(*=======================================================*)
	INIT:
		IF fb_state_entry.E THEN
			fb_ton_wz.IN := FALSE;
			fb_ton_uez.IN := FALSE;
			fb_ton_quitt.IN := FALSE;
			st_ctrl_out.b_fehler := FALSE;
			st_ctrl_out.b_bereit := FALSE;
			st_ctrl_out.b_fertig := FALSE;
			st_ctrl_out.b_kontroller_start := FALSE;
			zyl_wt_zentrierer_tisch.st_ctrl.in.b_einfahren := FALSE;
			zyl_wt_zentrierer_tisch.st_ctrl.in.b_ausfahren := FALSE;
			zyl_wt_zentrierer_tisch.st_ctrl.in.b_luftlos := FALSE;
			axis_transport_wt_achse.st_ctrl.in.b_start := FALSE;
			axis_z_achse.st_ctrl.in.b_start := FALSE;
			stueckzahlen.st_ctrl.in.b_gutteil_produziert := FALSE;
			sm_wt_hat_beladepos_nicht_verlassen := FALSE;
			sm_tagnummer_ungueltig := FALSE;
			sm_wt_hat_kein_tag := FALSE;
			sm_tagreader_nicht_fertig := FALSE;
			sm_keine_bandfreigabe := FALSE;
			bm_abfrage_wt_auf_beladepos := FALSE;
			bm_warte_auf_wt_an_stopper := FALSE;
			balluff_tag_reader.st_ctrl.in.b_start_lesen := FALSE;
			balluff_tag_reader.st_ctrl.in.b_start_schreiben := FALSE;
			zyl_Indexier_Bestueckpos.st_ctrl.in.b_ausfahren := FALSE;
			zyl_Indexier_Bestueckpos.st_ctrl.in.b_einfahren := FALSE;
			bMerkerSchrittketteKommtVonInit := TRUE;
		END_IF

		(*-----------------------Weiterschaltbedingungen----------------------------*)
		IF st_ctrl_in.b_init THEN
			zyl_wt_zentrierer_tisch.st_ctrl.in.b_quittieren := FALSE;
			zyl_Indexier_Bestueckpos.st_ctrl.in.b_quittieren := FALSE;
			fb_state_entry.i16_next_step := 20;
		END_IF

(*=======================================================*)
	20: fb_state_entry.s_debugtext := 'Initialisierung: Stopper an Bestücktisch ausfahren und Zentrierer einfahren';

		(*-----------------------Weiterschaltbedingungen----------------------------*)
		IF e_wt_im_aktionsfeld THEN
			fb_state_entry.i16_next_step := 25;
		ELSE
			fb_state_entry.i16_next_step := 22;
		END_IF

(*=======================================================*)
	22: fb_state_entry.s_debugtext := 'Initialisierung: Stopper an Bestücktisch ausfahren und Zentrierer einfahren';

		IF fb_state_entry.E THEN
			zyl_wt_zentrierer_tisch.st_ctrl.in.b_einfahren := TRUE;
		END_IF

		(*-----------------------Weiterschaltbedingungen----------------------------*)
		IF  zyl_wt_zentrierer_tisch.st_ctrl.out.b_eingefahren THEN
			zyl_wt_zentrierer_tisch.st_ctrl.in.b_einfahren := FALSE;
			fb_state_entry.i16_next_step := 30;
		END_IF

(*=======================================================*)
	25: fb_state_entry.s_debugtext := 'Initialisierung: Stopper an Bestücktisch ausfahren und Zentrierer einfahren';

		IF fb_state_entry.E THEN
			zyl_wt_zentrierer_tisch.st_ctrl.in.b_ausfahren := TRUE;
		END_IF

		(*-----------------------Weiterschaltbedingungen----------------------------*)
		IF  zyl_wt_zentrierer_tisch.st_ctrl.out.b_ausgefahren THEN
			zyl_wt_zentrierer_tisch.st_ctrl.in.b_ausfahren := FALSE;
			fb_state_entry.i16_next_step := 30;
		END_IF

(*=======================================================*)
	30: fb_state_entry.s_debugtext := 'Indexierzylinder wieder einfahren';

		IF fb_state_entry.E THEN
			zyl_Indexier_Bestueckpos.st_ctrl.in.b_ausfahren:= TRUE;
		END_IF

		(*-----------------------Weiterschaltbedingungen----------------------------*)
		IF zyl_Indexier_Bestueckpos.st_ctrl.out.b_ausgefahren THEN
			zyl_Indexier_Bestueckpos.st_ctrl.in.b_ausfahren:= FALSE;
			fb_state_entry.i16_next_step := 35;
		END_IF

(*=======================================================*)
	35: fb_state_entry.s_debugtext := 'warten auf Achse bereit';

		(*-----------------------Weiterschaltbedingungen----------------------------*)
		IF	axis_transport_wt_achse.st_ctrl.out.b_bereit AND
			NOT axis_transport_wt_achse.st_ctrl.in.b_start THEN
			fb_state_entry.i16_next_step := 40;
		END_IF

(*=======================================================*)
	40: fb_state_entry.s_debugtext := 'Fahre Achse wieder zurück';

		IF fb_state_entry.E THEN
			ST_WT_Transport_Achse.lr_Achspos_in:=gst_datensatz.st_md.st_md_transport_wt_achse.lr_startposition;
			ST_WT_Transport_Achse.lr_Velo_in:= gst_datensatz.st_md.r_geschwindigkeit_achse_transport;
			ST_WT_Transport_Achse.enu_cmd_in:=MOVE_ABSOLUTE;
			axis_transport_wt_achse.st_ctrl.in.b_start := TRUE;
		END_IF

		(*-----------------------Weiterschaltbedingungen----------------------------*)
		IF  axis_transport_wt_achse.st_ctrl.out.b_busy THEN
			axis_transport_wt_achse.st_ctrl.in.b_start := FALSE;
			fb_state_entry.i16_next_step := 50;
		END_IF

(*=======================================================*)
	50: fb_state_entry.s_debugtext := 'warten auf Achse hinten fertig';

		(*-----------------------Weiterschaltbedingungen----------------------------*)
		IF	axis_transport_wt_achse.st_ctrl.out.b_fertig  THEN
			fb_state_entry.i16_next_step := BEREIT;
		END_IF

(*=======================================================*)
	BEREIT:	fb_state_entry.s_debugtext := 'Warte auf Start von Kontroller';

		IF fb_state_entry.E THEN
			st_ctrl_out.b_bereit := TRUE;
			st_ctrl_out.b_fertig := TRUE;
			stueckzahlen.st_ctrl.in.b_gutteil_produziert := FALSE;
		END_IF

		(*-----------------------Weiterschaltbedingungen----------------------------*)
		IF st_config.b_station_aktiv OR st_config.b_station_in_simulation THEN

		(* WT Transport aktiv oder in Simulation *)
			IF 	st_ctrl_in.b_start  AND
				((NOT ST_Virtuelle_Masterachse.b_merker_bandende_links  AND
 				NOT ST_Virtuelle_Masterachse.b_merker_bandende_rechts) OR
				gst_datensatz.st_md.b_auto_Bandwechsel) THEN
			(* WT Transport gestartet *)
				st_ctrl_out.b_fertig := FALSE;
				fb_ton_wz.IN := FALSE;
				st_ctrl_out.b_kontroller_start := TRUE;
				(* Abfrage, ob Schrittkette von Init kommt und ob WT auf Beladepos ist *)
				IF bMerkerSchrittketteKommtVonInit AND
					e_wt_auf_beladepos THEN
					fb_state_entry.i16_next_step := 150;	(* WT auslesen und prüfen, ob dieser schon bestückt wurde *)
				ELSE
					fb_state_entry.i16_next_step := 110;
				END_IF
			END_IF

		(* WT-Transport nicht aktiv  *)
		ELSE
			IF fb_r_trig_start.Q THEN
				(* Nur Z-Achse gestartet *)
				st_ctrl_out.b_fertig := FALSE;
				fb_ton_wz.IN := FALSE;
				fb_state_entry.i16_next_step := 500;
			END_IF
		END_IF

		IF fb_state_entry.X THEN
			bMerkerSchrittketteKommtVonInit := FALSE;
		END_IF

(*=======================================================*)
	110: fb_state_entry.s_debugtext := 'WT-Abfrage auf Beladeposition';

		IF fb_state_entry.E THEN
			bm_abfrage_wt_auf_beladepos := TRUE;
		END_IF

		(*-----------------------Weiterschaltbedingungen----------------------------*)
		IF e_wt_im_aktionsfeld THEN
			(* Ein WT ist anwesend zum rausschicken *)
			IF NOT ST_WT_Transport_Abgabe.e_wt_auf_abgabepos THEN
				(* Erst wenn kein Stau vorhanden ist, dann wird der WT weiter gelassen *)
				fb_state_entry.i16_next_step := 115;
			END_IF
		ELSE	(* Kein WT da, deshalb einen holen *)
			fb_state_entry.i16_next_step := 130;
		END_IF

		IF fb_state_entry.X THEN
			bm_abfrage_wt_auf_beladepos := FALSE;
			st_ctrl_out.b_kontroller_start := FALSE;
		END_IF

(*=======================================================*)
	115: fb_state_entry.s_debugtext := 'Indexierzylinder Bestückposition ausfahren (WT festhalten)';

		IF fb_state_entry.E THEN
			zyl_Indexier_Bestueckpos.st_ctrl.in.b_einfahren:= TRUE;
		END_IF

		(*-----------------------Weiterschaltbedingungen----------------------------*)
		IF zyl_Indexier_Bestueckpos.st_ctrl.out.b_eingefahren THEN
			zyl_Indexier_Bestueckpos.st_ctrl.in.b_einfahren:= FALSE;
			fb_state_entry.i16_next_step := 120;
		END_IF

(*=======================================================*)
	120: fb_state_entry.s_debugtext := 'WT-Zentrierer einfahren';

		IF fb_state_entry.E THEN
			zyl_wt_zentrierer_tisch.st_ctrl.in.b_einfahren := TRUE;
			fb_Zentrierer_einfahren(b_start:= TRUE, t_zeit=> );
		END_IF

		(*-----------------------Weiterschaltbedingungen----------------------------*)
		IF zyl_wt_zentrierer_tisch.st_ctrl.out.b_eingefahren THEN
			zyl_wt_zentrierer_tisch.st_ctrl.in.b_einfahren := FALSE;
			fb_Zentrierer_einfahren(b_start:= FALSE, t_zeit=>t_Zentrierer_einfahren);
			fb_state_entry.i16_next_step := 130;
		END_IF

(*=======================================================*)
	130: fb_state_entry.s_debugtext := 'WT ist auf Warteposition und mit Indexierzylinder fixiert, wenn 2 Sekunden kein WT aus der vorherigen Zelle kommt wird der WT weitergeschickt';

		IF fb_state_entry.E THEN
			bm_abfrage_wt_auf_wartepos := TRUE;
		END_IF

		(*-----------------------Weiterschaltbedingungen----------------------------*)
		IF ST_WT_Transport_Warteposition_1700.e_wt_auf_wartepos_1700 AND
			 zyl_Indexier_Einlauf.st_ctrl.out.b_eingefahren AND
			ST_WT_Transport_Warteposition_1700.b_helpStartAchse AND
			zyl_wt_stopper_tisch.st_ctrl.out.b_eingefahren THEN
			fb_state_entry.i16_next_step := 135;
		ELSIF fb_state_entry.fb_ton_Step.ET >= T#2S AND
			 zyl_Indexier_Bestueckpos.st_ctrl.out.b_eingefahren THEN
			fb_state_entry.i16_next_step := 132;
		END_IF

(*=======================================================*)
	132: fb_state_entry.s_debugtext := 'Warten bis kein WT mehr auf der Abgabeposition steht';

		(*-----------------------Weiterschaltbedingungen----------------------------*)
		IF NOT ST_WT_Transport_Abgabe.e_wt_auf_abgabepos THEN
			fb_state_entry.i16_next_step := 135;
		END_IF

(*=======================================================*)
	135: fb_state_entry.s_debugtext := 'warten auf Achse bereit';

		(*-----------------------Weiterschaltbedingungen----------------------------*)
		IF	axis_transport_wt_achse.st_ctrl.out.b_bereit AND
			NOT axis_transport_wt_achse.st_ctrl.out.b_busy  AND
			NOT axis_transport_wt_achse.st_ctrl.in.b_start AND
			((ST_WT_Transport_Warteposition_1700.b_helpStartAchse AND
			ST_WT_Transport_Warteposition_1700.e_wt_auf_wartepos_1700)
			OR
			(zyl_Indexier_Einlauf.st_ctrl.out.b_ausgefahren AND
			NOT ST_WT_Transport_Warteposition_1700.e_wt_auf_wartepos_1700))  THEN
			fb_state_entry.i16_next_step := 140;
		END_IF

(*=======================================================*)
	140: fb_state_entry.s_debugtext := 'Fahre Achse nach vorne -> Bestückposition';

		IF fb_state_entry.E THEN
			ST_WT_Transport_Achse.lr_Achspos_in:=gst_datensatz.st_md.st_md_transport_wt_achse.lr_wt_uebergabepos;
			ST_WT_Transport_Achse.lr_Velo_in:= gst_datensatz.st_md.r_geschwindigkeit_achse_transport;
			ST_WT_Transport_Achse.enu_cmd_in:=MOVE_ABSOLUTE;
			axis_transport_wt_achse.st_ctrl.in.b_start := TRUE;

			st_ctrl_out.b_kontroller_start := TRUE;
		END_IF

		(*-----------------------Weiterschaltbedingungen----------------------------*)
		IF	axis_transport_wt_achse.st_ctrl.out.b_busy THEN
			axis_transport_wt_achse.st_ctrl.in.b_start := FALSE;
			fb_state_entry.i16_next_step := 145;
		END_IF

(*=======================================================*)
	145: fb_state_entry.s_debugtext := 'warten auf Achse vorne fertig';

		(*-----------------------Weiterschaltbedingungen----------------------------*)
		IF	axis_transport_wt_achse.st_ctrl.out.b_fertig THEN
			IF  zyl_Indexier_Einlauf.st_ctrl.out.b_eingefahren THEN
				fb_state_entry.i16_next_step := 147;	(* Neuer WT kommt von Warteposition *)
			ELSE
				fb_state_entry.i16_next_step := 300;	(* Es kommt kein neuer WT *)
			END_IF
		END_IF

		IF fb_state_entry.X THEN
			st_ctrl_out.b_kontroller_start := FALSE;
		END_IF

(*=======================================================*)
	147: fb_state_entry.s_debugtext := 'Prüfe, ob WT auf Beladeposition angekommen ist';

		(*-----------------------Weiterschaltbedingungen----------------------------*)
		IF e_wt_im_aktionsfeld AND
			NOT  ST_WT_Transport_Warteposition_1700.e_wt_auf_wartepos_1700  THEN
			fb_state_entry.i16_next_step := 150;
		ELSE
			sm_wt_hat_beladepos_nicht_verlassen := TRUE;
			fb_state_entry.i16_next_step := FEHLER;
		END_IF

(*=======================================================*)
	150: (*erst weiter wenn Abgabe funktioniert hat  *)

		IF 	NOT ST_WT_Transport_Abgabe.sm_wt_hat_abgabepos_nicht_verlassen THEN
			fb_state_entry.i16_next_step := 152;
		END_IF

		IF fb_state_entry.fb_ton_Step.ET > t#5s  THEN
			fb_state_entry.i16_next_step := STOP;
		END_IF

(*=======================================================*)
	152: (* WT-Zentrierer ausfahren *)

		IF fb_state_entry.E THEN
			zyl_wt_zentrierer_tisch.st_ctrl.in.b_ausfahren := TRUE;
			zyl_Indexier_Bestueckpos.st_ctrl.in.b_ausfahren:= TRUE;
			fb_Zentrierer_ausfahren(b_start:= TRUE, t_zeit=> );
		END_IF

		(*-----------------------Weiterschaltbedingungen----------------------------*)
		IF zyl_wt_zentrierer_tisch.st_ctrl.out.b_ausgefahren AND
			NOT ST_TippTasten.b_einfaedeln_aktiv AND
			NOT ST_Virtuelle_Masterachse.b_merker_bandende_links  AND
 			NOT ST_Virtuelle_Masterachse.b_merker_bandende_rechts AND
			zyl_Indexier_Bestueckpos.st_ctrl.out.b_ausgefahren THEN
			fb_Zentrierer_ausfahren(b_start:= FALSE, t_zeit=> t_Zentrierer_ausfahren);
			zyl_wt_zentrierer_tisch.st_ctrl.in.b_ausfahren := FALSE;
			fb_state_entry.i16_next_step := 155;
		END_IF

(*=======================================================*)
	155: fb_state_entry.s_debugtext := 'WT-Tag mit RFID-Lesegerät abfragen';

		(*-----------------------Weiterschaltbedingungen----------------------------*)
		IF  fb_state_entry.fb_ton_Step.ET >= T#100MS THEN
			IF e_wt_im_aktionsfeld THEN
				(* Tag auslesen *)
				fb_state_entry.i16_next_step := 160;
			ELSE
				(* Kein Tag auf WT *)
				sm_wt_hat_kein_tag := TRUE;
				fb_state_entry.i16_next_step := FEHLER;
			END_IF
		END_IF

(*=======================================================*)
	160: fb_state_entry.s_debugtext := 'Prüfe ob Simulation';

		(*-----------------------Weiterschaltbedingungen----------------------------*)
		IF 	st_config.b_station_in_simulation AND
			NOT visu.b_inbetriebnahme THEN
			fb_state_entry.i16_next_step := 300;
		ELSE
			fb_state_entry.i16_next_step := 170;
		END_IF

(*=======================================================*)
	170: fb_state_entry.s_debugtext := 'Z-Achse und anschliessend Bestückachse wird gestartet';

		IF fb_state_entry.E THEN
			axis_z_achse.st_ctrl.in.b_start := TRUE;
			(*Zeitmessung Trägerwechsel stoppen und ausgeben*)
			fb_WT_WechselZeit(b_start:=FALSE , t_zeit=>t_WT_WechselZeit );
		END_IF

		(*-----------------------Weiterschaltbedingungen----------------------------*)
		IF axis_z_achse.st_ctrl.out.b_busy THEN
			axis_z_achse.st_ctrl.in.b_start := FALSE;
			fb_state_entry.i16_next_step := 175;
		END_IF

(*=======================================================*)
	175: (*erst weiter wenn Abgabe funktioniert hat  *)

		IF 	NOT ST_WT_Transport_Abgabe.sm_wt_hat_abgabepos_nicht_verlassen THEN
			fb_state_entry.i16_next_step := 180;
		END_IF

		IF fb_state_entry.fb_ton_Step.ET > t#5s  THEN
			fb_state_entry.i16_next_step := STOP;
		END_IF

(*=======================================================*)
	180: fb_state_entry.s_debugtext := 'Indexierzylinder wieder einfahren (WT freigeben)';

		IF fb_state_entry.E THEN
			zyl_Indexier_Bestueckpos.st_ctrl.in.b_ausfahren:= TRUE;
		END_IF

		(*-----------------------Weiterschaltbedingungen----------------------------*)
		IF zyl_Indexier_Bestueckpos.st_ctrl.out.b_ausgefahren AND
			zyl_Indexier_Einlauf.st_ctrl.out.b_ausgefahren THEN
			zyl_Indexier_Bestueckpos.st_ctrl.in.b_ausfahren:= FALSE;
			fb_state_entry.i16_next_step := 190;
		END_IF

(*=======================================================*)
	190: fb_state_entry.s_debugtext := 'warten auf Achse bereit';

		(*-----------------------Weiterschaltbedingungen----------------------------*)
		IF	axis_transport_wt_achse.st_ctrl.out.b_bereit AND
			NOT axis_transport_wt_achse.st_ctrl.out.b_busy  AND
			NOT axis_transport_wt_achse.st_ctrl.in.b_start THEN
			fb_state_entry.i16_next_step := 200;
		END_IF

(*=======================================================*)
	200: fb_state_entry.s_debugtext := 'Fahre Achse wieder zurück';

		IF fb_state_entry.E THEN
			ST_WT_Transport_Achse.lr_Achspos_in:=gst_datensatz.st_md.st_md_transport_wt_achse.lr_startposition;
			ST_WT_Transport_Achse.lr_Velo_in:= gst_datensatz.st_md.r_geschwindigkeit_achse_transport;
			ST_WT_Transport_Achse.enu_cmd_in:=MOVE_ABSOLUTE;
			axis_transport_wt_achse.st_ctrl.in.b_start := TRUE;
		END_IF

		(*-----------------------Weiterschaltbedingungen----------------------------*)
		IF	axis_transport_wt_achse.st_ctrl.out.b_busy  THEN
			axis_transport_wt_achse.st_ctrl.in.b_start := FALSE;
			fb_state_entry.i16_next_step := 210;
		END_IF

(*=======================================================*)
	210: fb_state_entry.s_debugtext := 'warten auf Achse hinten fertig';

		(*-----------------------Weiterschaltbedingungen----------------------------*)
		IF	axis_transport_wt_achse.st_ctrl.out.b_fertig  THEN
			fb_state_entry.i16_next_step := 220;
		END_IF

(*=======================================================*)
	220: fb_state_entry.s_debugtext := 'Indexierzylinder Bestückposition ausfahren (WT festhalten)';

		IF fb_state_entry.E THEN
			zyl_Indexier_Bestueckpos.st_ctrl.in.b_einfahren:= TRUE;
		END_IF

		(*-----------------------Weiterschaltbedingungen----------------------------*)
		IF zyl_Indexier_Bestueckpos.st_ctrl.out.b_eingefahren THEN
			zyl_Indexier_Bestueckpos.st_ctrl.in.b_einfahren:= FALSE;
			fb_state_entry.i16_next_step := 230;
		END_IF

(*=======================================================*)
	230: fb_state_entry.s_debugtext := 'Bestückachse ist fertig';

		(*-----------------------Weiterschaltbedingungen----------------------------*)
		IF axis_virt_master.st_ctrl.out.b_fertig THEN
			IF axis_z_achse.st_ctrl.out.b_fertig THEN
				(*Zeitmessung Trägerwechsel starten*)
				fb_WT_WechselZeit(b_start:=TRUE , t_zeit=> );
				(*Zeitmessung zusammenfassen*)
				t_bestueckzeit:=ST_Z_Achse.t_Bestueckung;
				t_traegerwechselzeit:=t_WT_WechselZeit + ST_Z_Achse.t_Z_Achse_einfahren + ST_Z_Achse.t_Z_Achse_ausfahren;
				t_komplett_zyklus:= t_traegerwechselzeit + t_bestueckzeit;

				stueckzahlen.st_ctrl.in.b_gutteil_produziert := TRUE;

				st_ctrl_out.b_kontroller_start := FALSE;
				fb_state_entry.i16_next_step := BEREIT;
			END_IF
		END_IF

(*=======================================================*)
	300: fb_state_entry.s_debugtext := 'Indexierzylinder wieder einfahren (WT freigeben)';

		IF fb_state_entry.E THEN
			zyl_Indexier_Bestueckpos.st_ctrl.in.b_ausfahren:= TRUE;
		END_IF

		(*-----------------------Weiterschaltbedingungen----------------------------*)
		IF zyl_Indexier_Bestueckpos.st_ctrl.out.b_ausgefahren AND
			zyl_Indexier_Einlauf.st_ctrl.out.b_ausgefahren THEN
			zyl_Indexier_Bestueckpos.st_ctrl.in.b_ausfahren:= FALSE;
			fb_state_entry.i16_next_step := 310;
		END_IF

(*=======================================================*)
	310: fb_state_entry.s_debugtext := 'warten auf Achse bereit';

		(*-----------------------Weiterschaltbedingungen----------------------------*)
		IF	axis_transport_wt_achse.st_ctrl.out.b_bereit AND
			NOT axis_transport_wt_achse.st_ctrl.out.b_busy  AND
			NOT axis_transport_wt_achse.st_ctrl.in.b_start THEN
			fb_state_entry.i16_next_step := 320;
		END_IF

(*=======================================================*)
	320: fb_state_entry.s_debugtext := 'Fahre Achse wieder zurück';

		IF fb_state_entry.E THEN
			ST_WT_Transport_Achse.lr_Achspos_in:=gst_datensatz.st_md.st_md_transport_wt_achse.lr_startposition;
			ST_WT_Transport_Achse.lr_Velo_in:= gst_datensatz.st_md.r_geschwindigkeit_achse_transport;
			ST_WT_Transport_Achse.enu_cmd_in:=MOVE_ABSOLUTE;
			axis_transport_wt_achse.st_ctrl.in.b_start := TRUE;
		END_IF

		(*-----------------------Weiterschaltbedingungen----------------------------*)
		IF	axis_transport_wt_achse.st_ctrl.out.b_busy  THEN
			axis_transport_wt_achse.st_ctrl.in.b_start := FALSE;
			fb_state_entry.i16_next_step := 330;
		END_IF

(*=======================================================*)
	330: fb_state_entry.s_debugtext := 'warten auf Achse hinten fertig';

		(*-----------------------Weiterschaltbedingungen----------------------------*)
		IF	axis_transport_wt_achse.st_ctrl.out.b_fertig  THEN
			fb_state_entry.i16_next_step := BEREIT;
		END_IF

(*=======================================================*)
	500: fb_state_entry.s_debugtext := 'Warte bis angekommen an Stopper';
		IF fb_state_entry.E THEN
			bm_warte_auf_wt_an_stopper := TRUE;
		END_IF

		IF e_wt_im_aktionsfeld AND NOT fb_ton_wz.Q THEN
			fb_ton_wz.PT := t#3s;
			fb_ton_wz.IN := TRUE;
		END_IF

		(*-----------------------Weiterschaltbedingungen----------------------------*)
		IF fb_ton_wt_auf_beladepos.Q THEN
			fb_ton_wz.IN := FALSE;
			fb_state_entry.i16_next_step := 510;
		END_IF

		(*Abfrage auf Sensorfehler des Beladepositionssensors *)
		IF NOT e_wt_im_aktionsfeld  AND fb_ton_wz.Q THEN
			sm_sensorfehler_beladepos := TRUE;
			fb_state_entry.i16_next_step := FEHLER;
		END_IF

(*=======================================================*)
	510: fb_state_entry.s_debugtext := 'WT-Zentrierer ausfahren';

		IF fb_state_entry.E THEN
			zyl_wt_zentrierer_tisch.st_ctrl.in.b_ausfahren := TRUE;
		END_IF

		(*-----------------------Weiterschaltbedingungen----------------------------*)
		IF zyl_wt_zentrierer_tisch.st_ctrl.out.b_ausgefahren  THEN
			zyl_wt_zentrierer_tisch.st_ctrl.in.b_ausfahren := FALSE;
			fb_state_entry.i16_next_step := 520;
		END_IF

(*=======================================================*)
	520:	fb_state_entry.s_debugtext := 'Produktion ohne aktiven WT Transport';

		IF fb_state_entry.E THEN
			axis_z_achse.st_ctrl.in.b_start := TRUE;
		END_IF

		(*-----------------------Weiterschaltbedingungen----------------------------*)
		IF axis_z_achse.st_ctrl.out.b_fertig AND NOT fb_state_entry.E THEN
			axis_z_achse.st_ctrl.in.b_start := FALSE;
			stueckzahlen.st_ctrl.in.b_gutteil_produziert := TRUE;
			IF NOT b_Dauertest_Achsen THEN
				fb_state_entry.i16_next_step := BEREIT;
			ELSE
				(* zum Testen der Achsen nach Tausch, Bestückbild "Becherspucken", WKZ ausgebaut, Vorschubkontrolle abeschaltet,
				Bit muss von Programmierer geforct werden, zum Beenden Schlüsselschalter auf HAND und Zelle neu starten *)
				fb_state_entry.i16_next_step := 500;	(* Dauertest *)
			END_IF
		END_IF

(*=======================================================*)
	FEHLER:
		IF fb_state_entry.E THEN
			st_ctrl_out.b_fehler := TRUE;
			fb_ton_quitt.IN := FALSE;
			zyl_wt_zentrierer_tisch.st_ctrl.in.b_quittieren := FALSE;
			zyl_Indexier_Bestueckpos.st_ctrl.in.b_quittieren := FALSE;
			(*ST_Markiere_WT_NIO();*)
		END_IF

		(*-----------------------Weiterschaltbedingungen----------------------------*)
		IF st_ctrl_in.b_quitt AND NOT fb_state_entry.E THEN
			st_ctrl_out.b_fehler := FALSE;
			zyl_wt_zentrierer_tisch.st_ctrl.in.b_quittieren := TRUE;
			zyl_Indexier_Bestueckpos.st_ctrl.in.b_quittieren := TRUE;
			fb_ton_quitt.IN := TRUE;
		END_IF

		IF fb_ton_quitt.Q THEN
			fb_ton_quitt.IN := FALSE;
			fb_state_entry.i16_next_step := INIT;
		END_IF

(*=======================================================*)
	STOP:
		IF fb_state_entry.E THEN
			fb_ton_quitt.IN := FALSE;
			st_ctrl_out.b_kontroller_start := FALSE;
			zyl_wt_zentrierer_tisch.st_ctrl.in.b_quittieren := FALSE;
			zyl_Indexier_Bestueckpos.st_ctrl.in.b_quittieren := FALSE;

			(*ST_Markiere_WT_NIO();*)
		END_IF

		(*-----------------------Weiterschaltbedingungen----------------------------*)
		IF st_ctrl_in.b_quitt AND NOT fb_state_entry.E THEN
			fb_ton_quitt.IN := TRUE;
			zyl_wt_zentrierer_tisch.st_ctrl.in.b_quittieren := TRUE;
			zyl_Indexier_Bestueckpos.st_ctrl.in.b_quittieren := TRUE;
		END_IF

		IF fb_ton_quitt.Q THEN
			fb_ton_quitt.IN := FALSE;
			fb_state_entry.i16_next_step := INIT;
		END_IF
END_CASE

fb_state_entry(
	i16_next_step:= ,
	i16_pos:= 2,
	s_debugtext:= ,
	E=> ,
	X=> ,
	i16_step=> ,
	i16_last_step=> );

fb_ton_abfrage_wt_auf_beladepos (IN:=bm_abfrage_wt_auf_beladepos,PT:=t#30s);
fb_ton_warte_auf_wt_an_stopper (IN:=bm_warte_auf_wt_an_stopper,PT:=t#30s);

IF st_config.b_config_fertig THEN
	(* Fehlermeldungen ab dem Startindex in das globale Störmeldungsarray schreiben *)
	garr_stoermeldungen[st_config.i16_meld_startindex + 0] := sm_wt_hat_beladepos_nicht_verlassen;
	garr_stoermeldungen[st_config.i16_meld_startindex + 1] := sm_tagnummer_ungueltig;
	garr_stoermeldungen[st_config.i16_meld_startindex + 2] := sm_wt_hat_kein_tag;
	garr_stoermeldungen[st_config.i16_meld_startindex + 3] := FALSE;
	garr_stoermeldungen[st_config.i16_meld_startindex + 4] := sm_tagreader_nicht_fertig;
	garr_stoermeldungen[st_config.i16_meld_startindex + 5] := sm_keine_bandfreigabe;
	garr_stoermeldungen[st_config.i16_meld_startindex + 6] := FALSE;
	garr_stoermeldungen[st_config.i16_meld_startindex + 7] := FALSE;
	garr_stoermeldungen[st_config.i16_meld_startindex + 8] := FALSE;
	garr_stoermeldungen[st_config.i16_meld_startindex + 9] := FALSE;
	garr_stoermeldungen[st_config.i16_meld_startindex + 10] := FALSE;
	garr_stoermeldungen[st_config.i16_meld_startindex + 11] := FALSE;
	garr_stoermeldungen[st_config.i16_meld_startindex + 12] := FALSE;
	garr_stoermeldungen[st_config.i16_meld_startindex + 13] := FALSE;
	garr_stoermeldungen[st_config.i16_meld_startindex + 14] := FALSE;
	garr_stoermeldungen[st_config.i16_meld_startindex + 15] := FALSE;
	garr_stoermeldungen[st_config.i16_meld_startindex + 16] := FALSE;
	garr_stoermeldungen[st_config.i16_meld_startindex + 17] := FALSE;
	garr_stoermeldungen[st_config.i16_meld_startindex + 18] := FALSE;
	garr_stoermeldungen[st_config.i16_meld_startindex + 19] := FALSE;
	
	garr_betriebsmeldungen[st_config.i16_meld_startindex + 0] := fb_ton_abfrage_wt_auf_beladepos.Q;
	garr_betriebsmeldungen[st_config.i16_meld_startindex + 1] := fb_ton_warte_auf_wt_an_stopper.Q;
	garr_betriebsmeldungen[st_config.i16_meld_startindex + 2] := FALSE;
	garr_betriebsmeldungen[st_config.i16_meld_startindex + 3] := FALSE;
	garr_betriebsmeldungen[st_config.i16_meld_startindex + 4] := FALSE;
	garr_betriebsmeldungen[st_config.i16_meld_startindex + 5] := FALSE;
	garr_betriebsmeldungen[st_config.i16_meld_startindex + 6] := FALSE;
	garr_betriebsmeldungen[st_config.i16_meld_startindex + 7] := FALSE;
	garr_betriebsmeldungen[st_config.i16_meld_startindex + 8] := FALSE;
	garr_betriebsmeldungen[st_config.i16_meld_startindex + 9] := FALSE;
	garr_betriebsmeldungen[st_config.i16_meld_startindex + 10] := FALSE;
	garr_betriebsmeldungen[st_config.i16_meld_startindex + 11] := FALSE;
	garr_betriebsmeldungen[st_config.i16_meld_startindex + 12] := FALSE;
	garr_betriebsmeldungen[st_config.i16_meld_startindex + 13] := FALSE;
	garr_betriebsmeldungen[st_config.i16_meld_startindex + 14] := FALSE;
	garr_betriebsmeldungen[st_config.i16_meld_startindex + 15] := FALSE;
	garr_betriebsmeldungen[st_config.i16_meld_startindex + 16] := FALSE;
	garr_betriebsmeldungen[st_config.i16_meld_startindex + 17] := FALSE;
	garr_betriebsmeldungen[st_config.i16_meld_startindex + 18] := FALSE;
	garr_betriebsmeldungen[st_config.i16_meld_startindex + 19] := FALSE;
END_IF
END_PROGRAM

(* POU Maschine1700/ST_Stoerungen_Quitt_1700, ST *)
PROGRAM ST_Stoerungen_Quitt_1700
VAR_INPUT
	st_config					: struct_config;
	st_ctrl_in					: struct_ctrl_in;
END_VAR
VAR_IN_OUT
	st_visu					: struct_visu;
	st_visu_hinten				: struct_visu_hinten;
END_VAR
VAR_OUTPUT
	st_ctrl_out				: struct_ctrl_out;
	b_lampe_stoerung		: BOOL;
	b_lampe_produktion		: BOOL;
END_VAR
VAR
	fb_ton_quitt				: TON;
	b_Merker_quitt			: BOOL:=FALSE;
	fb_ton_wz				: TON;
	fb_r_trig_quittieren			: R_TRIG;
	fb_state_entry				: ST_StateEntry;

	fb_blinker				: ST_Blinker;

	bm_Maschine_in_Gst		: BOOL := FALSE;
	bm_Check		: BOOL := FALSE;
	sm_disable_auto_reset	: BOOL := FALSE;
END_VAR
(* Zeiten *)
fb_ton_quitt(IN:= , PT:= t#300ms, Q=> , ET=> );
fb_ton_wz(IN:= , PT:= t#3000ms, Q=> , ET=> );

(* Flanken *)
fb_r_trig_quittieren(CLK:= (st_visu.b_quittieren OR st_visu_hinten.out.b_quittieren) AND gi16_betriebsart <> HAND, Q=> );

(* Blinker *)
fb_blinker(
	b_start:= TRUE,
	t_taktzeit_on:=t#500ms,
	t_taktzeit_off:=t#500ms,
	b_blinker_out=> );

(* Lampen *)
b_lampe_stoerung := gi16_maschinenstatusinfo = KEIN_STATUS OR gi16_maschinenstatusinfo = STATUS_FEHLER;

b_lampe_produktion := (fb_blinker.b_blinker_out AND
					(gi16_maschinenstatusinfo = STATUS_FEHLER_QUITTIERT OR
					gi16_maschinenstatusinfo = STATUS_BETRIEBSBEREIT)) OR
					gi16_maschinenstatusinfo = STATUS_MASCHINE_ARBEITET;

bm_Check:=(
	CheckBounds_ErrCnt+
	CheckByteZeroDiv_ErrCnt+
	CheckDWordZeroDiv_ErrCnt+
	CheckRealZeroDiv_ErrCnt+
	CheckWordZeroDiv_ErrCnt+
	CheckRangeSigned_ErrCnt+
	CheckRangeUnsigned_ErrCnt) > 0 ;

(* Toplevel *)
(* Hier nur Abschaltungen welche zu sofortigem Stop führen müssen *)
IF fb_state_entry.i16_step < FEHLER AND
	(axis_virt_master.st_ctrl.out.b_fehler OR
	axis_bestueckachse.st_ctrl.out.b_fehler OR
	axis_z_achse.st_ctrl.out.b_fehler OR
	axis_y_achse.st_ctrl.out.b_fehler OR
	ST_TouchProbe.st_ctrl_out.b_fehler OR
	(axis_bandeinzug_achse.st_ctrl.out.b_fehler AND gst_datensatz.st_wkz.i16_typ_bandeinzug = SERVO) OR
	bandspruehoeler.st_ctrl.out.b_fehler OR
	(bandeinzug_kontroller.st_ctrl.out.b_fehler AND gst_datensatz.st_wkz.i16_typ_bandeinzug = BANDWECHSLER_V2) OR
	bandwechsel_kontroller.st_ctrl.out.b_fehler OR
	wkz_absicherung.st_ctrl.out.b_fehler OR
	wt_transport_kontroller.st_ctrl.out.b_fehler OR
	balluff_tag_reader.st_ctrl.out.b_fehler OR
	haspel_kontroller.st_ctrl.out.b_fehler OR
	bbgen.st_ctrl.out.b_fehler OR
	wartung.st_ctrl.out.b_fehler OR
	betriebsfreigaben.st_ctrl.out.b_fehler OR
	einpresskraft_kontroller.st_ctrl.out.b_fehler OR
	safety.st_ctrl.out.b_fehler OR
	edit_mfps.st_ctrl.out.b_fehler OR
	Lesen_Schreiben_Tag.st_ctrl.out.b_fehler OR
	Service.st_ctrl.out.b_fehler OR
	axis_transport_wt_achse.st_ctrl.out.b_fehler)
	THEN
		fb_state_entry.i16_next_step := FEHLER;
END_IF

(* Prüfe ob BA = Hand -> Stoppe Abläufe *)
IF  fb_state_entry.i16_step > INIT  AND fb_state_entry.i16_step < FEHLER  AND gi16_betriebsart = HAND THEN
	fb_state_entry.i16_next_step := FEHLER;
END_IF

(* ======================================Schrittkette======================================== *)
fb_state_entry(
	i16_next_step:= ,
	i16_pos:= 1,
	s_debugtext:= ,
	E=> ,
	X=> ,
	i16_step=> ,
	i16_last_step=> );

CASE fb_state_entry.i16_step OF
(*=======================================================*)
	INIT_OBJ:
		IF st_config.b_config_fertig THEN
			fb_state_entry.i16_next_step := FEHLER;
		END_IF

(*=======================================================*)
	INIT:
		IF fb_state_entry.E THEN
			gi16_maschinenstatusinfo := STATUS_FEHLER_QUITTIERT;
			fb_ton_quitt.IN := FALSE;
			UPS.st_ctrl.in.b_quitt := FALSE;
			betriebsfreigaben.st_ctrl.in.b_quitt := FALSE;
			bandeinzug_kontroller.st_ctrl.in.b_quitt := FALSE;
			bandwechsel_kontroller.st_ctrl.in.b_quitt := FALSE;
			axis_virt_master.st_ctrl.in.b_quitt := FALSE;
			axis_bestueckachse.st_ctrl.in.b_quitt := FALSE;
			axis_y_achse.st_ctrl.in.b_quitt := FALSE;
			axis_z_achse.st_ctrl.in.b_quitt := FALSE;
			ST_TouchProbe.st_ctrl_in.b_quitt := FALSE;
			axis_bandeinzug_achse.st_ctrl.in.b_quitt := FALSE;
			bandspruehoeler.st_ctrl.in.b_quitt := FALSE;
			haspel_kontroller.st_ctrl.in.b_quitt := FALSE;
			hublift_links.st_ctrl.in.b_quitt := FALSE;
			hublift_rechts.st_ctrl.in.b_quitt := FALSE;
			wt_transport_kontroller.st_ctrl.in.b_quitt := FALSE;
			wkz_absicherung.st_ctrl.in.b_quitt := FALSE;
			stueckzahlen.st_ctrl.in.b_quitt := FALSE;
			balluff_tag_reader.st_ctrl.in.b_quitt := FALSE;
			bbgen.st_ctrl.in.b_quitt := FALSE;
			wartung.st_ctrl.in.b_quitt := FALSE;
			einpresskraft_kontroller.st_ctrl.in.b_quitt := FALSE;
			safety.st_ctrl.in.b_quitt := FALSE;
			edit_mfps.st_ctrl.in.b_quitt := FALSE;
			routing_backpanel.st_ctrl.in.b_quitt := FALSE;
			routing_nachbarpc.st_ctrl.in.b_quitt := FALSE;
			bm_Maschine_in_Gst := FALSE;
			Lesen_Schreiben_Tag.st_ctrl.in.b_quitt := FALSE;
			Service.st_ctrl.in.b_quitt := FALSE;
			ST_TippTasten.b_initialisierungsphase := TRUE;
			sm_disable_auto_reset := FALSE;
			axis_transport_wt_achse.st_ctrl.in.b_quitt := FALSE;
		END_IF

		(*-----------------------Weiterschaltbedingungen----------------------------*)
		IF safety.st_ctrl.out.b_bereit THEN
			fb_state_entry.i16_next_step := 11;
		END_IF

(*=======================================================*)
	11:
		IF fb_state_entry.E THEN
			axis_virt_master.st_ctrl.in.b_preinit := TRUE;
		END_IF

		(*-----------------------Weiterschaltbedingungen----------------------------*)
		IF axis_virt_master.st_ctrl.out.b_prebereit  THEN
			axis_virt_master.st_ctrl.in.b_preinit := FALSE;
			fb_state_entry.i16_next_step := 12;
		END_IF

(*=======================================================*)
	12:
		IF fb_state_entry.E THEN
			axis_z_achse.st_ctrl.in.b_preinit := TRUE;
		END_IF

		(*-----------------------Weiterschaltbedingungen----------------------------*)
		IF axis_z_achse.st_ctrl.out.b_prebereit  THEN
			axis_z_achse.st_ctrl.in.b_preinit := FALSE;
			fb_state_entry.i16_next_step := 13;
		END_IF

(*=======================================================*)
	13:
		IF fb_state_entry.E THEN
			axis_y_achse.st_ctrl.in.b_preinit := TRUE;
		END_IF

		(*-----------------------Weiterschaltbedingungen----------------------------*)
		IF axis_y_achse.st_ctrl.out.b_prebereit  THEN
			axis_y_achse.st_ctrl.in.b_preinit := FALSE;
			fb_state_entry.i16_next_step := 14;
		END_IF

(*=======================================================*)
	14:
		CASE gst_datensatz.st_wkz.i16_typ_bandeinzug OF
			BANDWECHSLER_V2:
				fb_state_entry.i16_next_step := 15;
			SERVO:
				IF fb_state_entry.E THEN
					axis_bandeinzug_achse.st_ctrl.in.b_preinit := TRUE;
				END_IF

				(*-----------------------Weiterschaltbedingungen----------------------------*)
				IF axis_bandeinzug_achse.st_ctrl.out.b_prebereit  THEN
					axis_bandeinzug_achse.st_ctrl.in.b_preinit := FALSE;
					fb_state_entry.i16_next_step := 15;
				END_IF
		END_CASE

(*=======================================================*)
	15:
		IF fb_state_entry.E THEN
			axis_bestueckachse.st_ctrl.in.b_preinit := TRUE;
		END_IF

		(*-----------------------Weiterschaltbedingungen----------------------------*)
		IF axis_bestueckachse.st_ctrl.out.b_prebereit  THEN
			axis_bestueckachse.st_ctrl.in.b_preinit := FALSE;
			fb_state_entry.i16_next_step := 16;
		END_IF

(*=======================================================*)
	16:
		(*Wenn die Bestückachse nicht in einem bestimmten Bereich steht, dann muss sie von Hand
		    freigefahren werden. Außer es ist die Nocke auf 0,0 gestellt*)
		IF	gst_datensatz.st_wkz.nockenschaltwerk_bestueckachse.arr_nocken[SP_DISABLE_AUTO_RESET].r_cam_begin = 0 AND
			gst_datensatz.st_wkz.nockenschaltwerk_bestueckachse.arr_nocken[SP_DISABLE_AUTO_RESET].r_cam_end = 0 THEN
				fb_state_entry.i16_next_step := 17;
		ELSE
			IF gst_datensatz.st_wkz.nockenschaltwerk_bestueckachse.arr_nocken[SP_DISABLE_AUTO_RESET].r_cam_begin > gst_datensatz.st_wkz.nockenschaltwerk_bestueckachse.arr_nocken[SP_DISABLE_AUTO_RESET].r_cam_end THEN
				IF bestueckachse.NcToPlc.ModuloActPos > gst_datensatz.st_wkz.nockenschaltwerk_bestueckachse.arr_nocken[SP_DISABLE_AUTO_RESET].r_cam_begin OR
					bestueckachse.NcToPlc.ModuloActPos < gst_datensatz.st_wkz.nockenschaltwerk_bestueckachse.arr_nocken[SP_DISABLE_AUTO_RESET].r_cam_end THEN
					sm_disable_auto_reset := TRUE;
					fb_state_entry.i16_next_step := FEHLER;
				ELSE
					fb_state_entry.i16_next_step := 17;
				END_IF
			ELSE
				IF bestueckachse.NcToPlc.ModuloActPos > gst_datensatz.st_wkz.nockenschaltwerk_bestueckachse.arr_nocken[SP_DISABLE_AUTO_RESET].r_cam_begin AND
					bestueckachse.NcToPlc.ModuloActPos < gst_datensatz.st_wkz.nockenschaltwerk_bestueckachse.arr_nocken[SP_DISABLE_AUTO_RESET].r_cam_end THEN
					sm_disable_auto_reset := TRUE;
					fb_state_entry.i16_next_step := FEHLER;
				ELSE
					fb_state_entry.i16_next_step := 17;
				END_IF
			END_IF
		END_IF
(*=======================================================*)
	17:
		(*-----------------------Weiterschaltbedingungen----------------------------*)
		IF 	gst_datensatz.st_md.b_anwahl_transport_achse  THEN
			fb_state_entry.i16_next_step := 18;
		ELSE
			fb_state_entry.i16_next_step := 20;
		END_IF

(*=======================================================*)
	18:
		IF fb_state_entry.E THEN
			axis_transport_wt_achse.st_ctrl.in.b_preinit := TRUE;
		END_IF

		(*-----------------------Weiterschaltbedingungen----------------------------*)
		IF axis_transport_wt_achse.st_ctrl.out.b_prebereit  THEN
			axis_transport_wt_achse.st_ctrl.in.b_preinit := FALSE;
			fb_state_entry.i16_next_step := 20;
		END_IF

(*=======================================================*)
	20:
		IF fb_state_entry.E THEN
			haspel_kontroller.st_ctrl.in.b_init := TRUE;
			bandspruehoeler.st_ctrl.in.b_init := TRUE;
			wkz_absicherung.st_ctrl.in.b_init := TRUE;
			stueckzahlen.st_ctrl.in.b_init := TRUE;
			(*balluff_tag_reader.st_ctrl.in.b_init := TRUE;*)
			einpresskraft_kontroller.st_ctrl.in.b_init := TRUE;
			edit_mfps.st_ctrl.in.b_init := TRUE;
		END_IF

		(*-----------------------Weiterschaltbedingungen----------------------------*)
		IF 	haspel_kontroller.st_ctrl.out.b_bereit  AND
			bandspruehoeler.st_ctrl.out.b_bereit  AND
			wkz_absicherung.st_ctrl.out.b_bereit AND
			einpresskraft_kontroller.st_ctrl.out.b_bereit AND
			balluff_tag_reader.st_ctrl.out.b_bereit AND
			edit_mfps.st_ctrl.out.b_bereit
			THEN
				haspel_kontroller.st_ctrl.in.b_init := FALSE;
				bandspruehoeler.st_ctrl.in.b_init := FALSE;
				wkz_absicherung.st_ctrl.in.b_init := FALSE;
				stueckzahlen.st_ctrl.in.b_init := FALSE;
				(*balluff_tag_reader.st_ctrl.in.b_init := FALSE;*)
				einpresskraft_kontroller.st_ctrl.in.b_init := FALSE;
				edit_mfps.st_ctrl.in.b_init := FALSE;
				fb_state_entry.i16_next_step := 30;
		END_IF

(*=======================================================*)
	30:
		CASE gst_datensatz.st_wkz.i16_typ_bandeinzug OF
			BANDWECHSLER_V2:
				IF fb_state_entry.E THEN
					bandeinzug_kontroller.st_ctrl.in.b_init := TRUE;
				END_IF
		
				(*-----------------------Weiterschaltbedingungen----------------------------*)
				IF bandeinzug_kontroller.st_ctrl.out.b_bereit THEN
					bandeinzug_kontroller.st_ctrl.in.b_init := FALSE;
					fb_state_entry.i16_next_step := 40;
				END_IF
			SERVO:
				fb_state_entry.i16_next_step := 40;
		END_CASE

(*=======================================================*)
	40:
		IF fb_state_entry.E THEN
			bandwechsel_kontroller.st_ctrl.in.b_init := TRUE;
		END_IF

		(*-----------------------Weiterschaltbedingungen----------------------------*)
		IF bandwechsel_kontroller.st_ctrl.out.b_bereit THEN
			bandwechsel_kontroller.st_ctrl.in.b_init := FALSE;
			fb_state_entry.i16_next_step := 50;
		END_IF

(*=======================================================*)
	50:
		IF fb_state_entry.E THEN
			axis_bestueckachse.st_ctrl.in.b_init := TRUE;
		END_IF

		(*-----------------------Weiterschaltbedingungen----------------------------*)
		IF axis_bestueckachse.st_ctrl.out.b_bereit  THEN
			axis_bestueckachse.st_ctrl.in.b_init := FALSE;
			fb_state_entry.i16_next_step := 60;
		END_IF

(*=======================================================*)
	60:
		CASE gst_datensatz.st_wkz.i16_typ_bandeinzug OF
			BANDWECHSLER_V2:
				IF fb_state_entry.E THEN
					axis_z_achse.st_ctrl.in.b_init := TRUE;
					axis_y_achse.st_ctrl.in.b_init := TRUE;
					axis_transport_wt_achse.st_ctrl.in.b_init := gst_datensatz.st_md.b_anwahl_transport_achse;
				END_IF
		
				(*-----------------------Weiterschaltbedingungen----------------------------*)
				IF 	axis_z_achse.st_ctrl.out.b_bereit AND
					axis_y_achse.st_ctrl.out.b_bereit AND
					(axis_transport_wt_achse.st_ctrl.out.b_bereit OR NOT gst_datensatz.st_md.b_anwahl_transport_achse)
					THEN
						axis_z_achse.st_ctrl.in.b_init := FALSE;
						axis_y_achse.st_ctrl.in.b_init := FALSE;
						axis_transport_wt_achse.st_ctrl.in.b_init := FALSE;
						fb_state_entry.i16_next_step := 70;
				END_IF
			SERVO:
				IF fb_state_entry.E THEN
					axis_z_achse.st_ctrl.in.b_init := TRUE;
					axis_y_achse.st_ctrl.in.b_init := TRUE;
					axis_bandeinzug_achse.st_ctrl.in.b_init := TRUE;
				END_IF
		
				(*-----------------------Weiterschaltbedingungen----------------------------*)
				IF 	axis_z_achse.st_ctrl.out.b_bereit AND
					axis_y_achse.st_ctrl.out.b_bereit AND
					axis_bandeinzug_achse.st_ctrl.out.b_bereit
					THEN
						axis_z_achse.st_ctrl.in.b_init := FALSE;
						axis_y_achse.st_ctrl.in.b_init := FALSE;
						fb_state_entry.i16_next_step := 70;
				END_IF
		END_CASE

(*=======================================================*)
	70:
		IF fb_state_entry.E THEN
			axis_virt_master.st_ctrl.in.b_init := TRUE;
		END_IF

		(*-----------------------Weiterschaltbedingungen----------------------------*)
		IF axis_virt_master.st_ctrl.out.b_bereit  THEN
			axis_virt_master.st_ctrl.in.b_init := FALSE;
			fb_state_entry.i16_next_step := 80;
		END_IF

(*=======================================================*)
	80:
		IF fb_state_entry.E THEN
			hublift_links.st_ctrl.in.b_init := TRUE;
			hublift_rechts.st_ctrl.in.b_init := TRUE;
			wt_transport_kontroller.st_ctrl.in.b_init := TRUE;
			ST_TouchProbe.st_ctrl_in.b_init := TRUE;
		END_IF

		(*-----------------------Weiterschaltbedingungen----------------------------*)
		IF hublift_links.st_ctrl.out.b_bereit AND hublift_rechts.st_ctrl.out.b_bereit AND wt_transport_kontroller.st_ctrl.out.b_bereit AND
			ST_TouchProbe.st_ctrl_out.b_bereit THEN
			hublift_links.st_ctrl.in.b_init := FALSE;
			hublift_rechts.st_ctrl.in.b_init := FALSE;
			wt_transport_kontroller.st_ctrl.in.b_init := FALSE;
			ST_TouchProbe.st_ctrl_in.b_init := FALSE;
			fb_state_entry.i16_next_step := BEREIT;
		END_IF

(*=======================================================*)
	BEREIT:
		IF fb_state_entry.E THEN
			ST_TippTasten.b_initialisierungsphase  := FALSE;
			(* Setze Maschinenstatus *)
			bm_Maschine_in_Gst := TRUE;
		END_IF

		(*Beim Einfädeln muss der Status geändert werden, damit nicht
		ständig neue Maschinendaten erzeugt werden*)
		IF ST_TippTasten.b_einfaedeln_aktiv THEN
			gi16_maschinenstatusinfo := STATUS_MASCHINE_ARBEITET;
		ELSE
			gi16_maschinenstatusinfo := STATUS_BETRIEBSBEREIT;
		END_IF

		(*-----------------------Weiterschaltbedingungen----------------------------*)
		IF NOT wt_transport_kontroller.st_ctrl.out.b_fertig THEN
			bm_Maschine_in_Gst := FALSE;
			fb_state_entry.i16_next_step := 110;
		END_IF

(*=======================================================*)
	110: (* Produktion *)
		IF fb_state_entry.E THEN
			gi16_maschinenstatusinfo := STATUS_MASCHINE_ARBEITET;
		END_IF

		(*-----------------------Weiterschaltbedingungen----------------------------*)
		IF wt_transport_kontroller.st_ctrl.out.b_fertig THEN
			fb_state_entry.i16_next_step := BEREIT;
		END_IF

(*=======================================================*)
	FEHLER:
		IF fb_state_entry.E THEN
			gi16_maschinenstatusinfo := STATUS_FEHLER;
			bm_Maschine_in_Gst := FALSE;
			ST_TippTasten.b_initialisierungsphase  := FALSE;
			fb_ton_quitt.IN := FALSE;
			fb_ton_wz.IN:=FALSE;
			s_alte_artikelnummer := '';

			(* Schlecht Stueckzahl erhöhen *)
			IF fb_state_entry.i16_last_step = 110 THEN
				stueckzahlen.st_ctrl.in.b_schlechtteil_produziert := TRUE;
			END_IF

			UPS.st_ctrl.in.b_quitt := FALSE;
			betriebsfreigaben.st_ctrl.in.b_quitt := FALSE;
			bandeinzug_kontroller.st_ctrl.in.b_quitt := FALSE;
			bandwechsel_kontroller.st_ctrl.in.b_quitt := FALSE;
			axis_virt_master.st_ctrl.in.b_quitt := FALSE;
			axis_bestueckachse.st_ctrl.in.b_quitt := FALSE;
			axis_y_achse.st_ctrl.in.b_quitt := FALSE;
			axis_z_achse.st_ctrl.in.b_quitt := FALSE;
			ST_TouchProbe.st_ctrl_in.b_quitt := FALSE;
			axis_bandeinzug_achse.st_ctrl.in.b_quitt := FALSE;
			bandspruehoeler.st_ctrl.in.b_quitt := FALSE;
			haspel_kontroller.st_ctrl.in.b_quitt := FALSE;
			hublift_links.st_ctrl.in.b_quitt := FALSE;
			hublift_rechts.st_ctrl.in.b_quitt := FALSE;
			wt_transport_kontroller.st_ctrl.in.b_quitt := FALSE;
			wkz_absicherung.st_ctrl.in.b_quitt := FALSE;
			stueckzahlen.st_ctrl.in.b_quitt := FALSE;
			balluff_tag_reader.st_ctrl.in.b_quitt := FALSE;
			bbgen.st_ctrl.in.b_quitt := FALSE;
			wartung.st_ctrl.in.b_quitt := FALSE;
			einpresskraft_kontroller.st_ctrl.in.b_quitt := FALSE;
			safety.st_ctrl.in.b_quitt := FALSE;
			edit_mfps.st_ctrl.in.b_quitt := FALSE;
			routing_backpanel.st_ctrl.in.b_quitt := FALSE;
			routing_nachbarpc.st_ctrl.in.b_quitt := FALSE;
			Lesen_Schreiben_Tag.st_ctrl.in.b_quitt := FALSE;
			Service.st_ctrl.in.b_quitt := FALSE;
			axis_transport_wt_achse.st_ctrl.in.b_quitt := FALSE;

			axis_virt_master.st_ctrl.in.b_preinit := FALSE;
			axis_bestueckachse.st_ctrl.in.b_preinit := FALSE;
			axis_y_achse.st_ctrl.in.b_preinit := FALSE;
			axis_z_achse.st_ctrl.in.b_preinit := FALSE;
			axis_bandeinzug_achse.st_ctrl.in.b_preinit := FALSE;
			axis_transport_wt_achse.st_ctrl.in.b_preinit := FALSE;

			bandeinzug_kontroller.st_ctrl.in.b_init := FALSE;
			bandwechsel_kontroller.st_ctrl.in.b_init := FALSE;
			axis_virt_master.st_ctrl.in.b_init := FALSE;
			axis_bestueckachse.st_ctrl.in.b_init := FALSE;
			axis_y_achse.st_ctrl.in.b_init := FALSE;
			axis_z_achse.st_ctrl.in.b_init := FALSE;
			ST_TouchProbe.st_ctrl_in.b_init := FALSE;
			axis_bandeinzug_achse.st_ctrl.in.b_init := FALSE;
			bandspruehoeler.st_ctrl.in.b_init := FALSE;
			haspel_kontroller.st_ctrl.in.b_init := FALSE;
			hublift_links.st_ctrl.in.b_init := FALSE;
			hublift_rechts.st_ctrl.in.b_init := FALSE;
			wt_transport_kontroller.st_ctrl.in.b_init := FALSE;
			wkz_absicherung.st_ctrl.in.b_init := FALSE;
			stueckzahlen.st_ctrl.in.b_init := FALSE;
			(*balluff_tag_reader.st_ctrl.in.b_init := FALSE;*)
			edit_mfps.st_ctrl.in.b_init := FALSE;
			axis_transport_wt_achse.st_ctrl.in.b_init := FALSE;
		END_IF

		(* Fehlerhandling: was soll bei welchem Fehler passieren? *)
		IF 	NOT fb_ton_quitt.IN THEN
			(* Stoppe/Halte Komponenten an *)
			bandeinzug_kontroller.st_ctrl.in.b_stop := TRUE;
			bandwechsel_kontroller.st_ctrl.in.b_stop := TRUE;
			bandspruehoeler.st_ctrl.in.b_stop := TRUE;
			(*haspel_kontroller.st_ctrl.in.b_stop := TRUE;*)
			hublift_links.st_ctrl.in.b_stop := TRUE;
			hublift_rechts.st_ctrl.in.b_stop := TRUE;
			wt_transport_kontroller.st_ctrl.in.b_stop := TRUE;
			stueckzahlen.st_ctrl.in.b_stop := TRUE;
			balluff_tag_reader.st_ctrl.in.b_stop := TRUE;
			edit_mfps.st_ctrl.in.b_stop := TRUE;

			(* Diese Fehler führt zum "Stop" in der Maschine *)
			IF safety.st_ctrl.out.b_fehler THEN
				axis_virt_master.st_ctrl.in.b_stop := TRUE;
				axis_bestueckachse.st_ctrl.in.b_stop := TRUE;
				axis_z_achse.st_ctrl.in.b_stop := TRUE;
				axis_y_achse.st_ctrl.in.b_stop := TRUE;
				axis_bandeinzug_achse.st_ctrl.in.b_stop := TRUE;
				axis_transport_wt_achse.st_ctrl.in.b_stop := TRUE;
				axis_virt_master.st_ctrl.in.b_halt := FALSE;
				axis_bestueckachse.st_ctrl.in.b_halt := FALSE;
				axis_z_achse.st_ctrl.in.b_halt := FALSE;
				axis_y_achse.st_ctrl.in.b_halt := FALSE;
				axis_bandeinzug_achse.st_ctrl.in.b_halt := FALSE;
				axis_transport_wt_achse.st_ctrl.in.b_halt := FALSE;
			ELSE
				axis_virt_master.st_ctrl.in.b_halt := TRUE;
				axis_bestueckachse.st_ctrl.in.b_halt := TRUE;
				axis_z_achse.st_ctrl.in.b_halt := TRUE;
				axis_y_achse.st_ctrl.in.b_halt := TRUE;
				axis_bandeinzug_achse.st_ctrl.in.b_halt := TRUE;
				axis_transport_wt_achse.st_ctrl.in.b_halt := TRUE;
				axis_virt_master.st_ctrl.in.b_stop := FALSE;
				axis_bestueckachse.st_ctrl.in.b_stop := FALSE;
				axis_z_achse.st_ctrl.in.b_stop := FALSE;
				axis_y_achse.st_ctrl.in.b_stop := FALSE;
				axis_bandeinzug_achse.st_ctrl.in.b_stop := FALSE;
				axis_transport_wt_achse.st_ctrl.in.b_stop := FALSE;
			END_IF
		END_IF

		(*-----------------------Weiterschaltbedingungen----------------------------*)
		IF 	fb_r_trig_quittieren.Q THEN
			fb_ton_wz.IN:=TRUE;
			b_Merker_quitt:=TRUE;
		END_IF
		IF 	(b_Merker_quitt AND ST_Betriebsfreigaben.e_druckwaechter) OR
			fb_ton_wz.Q THEN
			fb_ton_wz.IN:=FALSE;
			b_Merker_quitt:=FALSE;
			fb_ton_quitt.IN := TRUE;
			(* QUITT *)
			UPS.st_ctrl.in.b_quitt := TRUE;
			betriebsfreigaben.st_ctrl.in.b_quitt := TRUE;
			bandeinzug_kontroller.st_ctrl.in.b_quitt := TRUE;
			bandwechsel_kontroller.st_ctrl.in.b_quitt := TRUE;
			axis_virt_master.st_ctrl.in.b_quitt := TRUE;
			axis_bestueckachse.st_ctrl.in.b_quitt := TRUE;
			axis_y_achse.st_ctrl.in.b_quitt := TRUE;
			axis_z_achse.st_ctrl.in.b_quitt := TRUE;
			ST_TouchProbe.st_ctrl_in.b_quitt := TRUE;
			axis_bandeinzug_achse.st_ctrl.in.b_quitt := TRUE;
			bandspruehoeler.st_ctrl.in.b_quitt := TRUE;
			haspel_kontroller.st_ctrl.in.b_quitt := TRUE;
			hublift_links.st_ctrl.in.b_quitt := TRUE;
			hublift_rechts.st_ctrl.in.b_quitt := TRUE;
			wt_transport_kontroller.st_ctrl.in.b_quitt := TRUE;
			wkz_absicherung.st_ctrl.in.b_quitt := TRUE;
			stueckzahlen.st_ctrl.in.b_quitt := TRUE;
			balluff_tag_reader.st_ctrl.in.b_quitt := TRUE;
			bbgen.st_ctrl.in.b_quitt := TRUE;
			wartung.st_ctrl.in.b_quitt := TRUE;
			einpresskraft_kontroller.st_ctrl.in.b_quitt := TRUE;
			safety.st_ctrl.in.b_quitt := TRUE;
			edit_mfps.st_ctrl.in.b_quitt := TRUE;
			routing_backpanel.st_ctrl.in.b_quitt := TRUE;
			routing_nachbarpc.st_ctrl.in.b_quitt := TRUE;
			Lesen_Schreiben_Tag.st_ctrl.in.b_quitt := TRUE;
			Service.st_ctrl.in.b_quitt := TRUE;
			axis_transport_wt_achse.st_ctrl.in.b_quitt := TRUE;
			(* STOP *)
			bandeinzug_kontroller.st_ctrl.in.b_stop := FALSE;
			bandwechsel_kontroller.st_ctrl.in.b_stop := FALSE;
			axis_virt_master.st_ctrl.in.b_stop := FALSE;
			axis_bestueckachse.st_ctrl.in.b_stop := FALSE;
			axis_y_achse.st_ctrl.in.b_stop := FALSE;
			axis_z_achse.st_ctrl.in.b_stop := FALSE;
			axis_bandeinzug_achse.st_ctrl.in.b_stop := FALSE;
			bandspruehoeler.st_ctrl.in.b_stop := FALSE;
			haspel_kontroller.st_ctrl.in.b_stop := FALSE;
			hublift_links.st_ctrl.in.b_stop := FALSE;
			hublift_rechts.st_ctrl.in.b_stop := FALSE;
			wt_transport_kontroller.st_ctrl.in.b_stop := FALSE;
			wkz_absicherung.st_ctrl.in.b_stop := FALSE;
			stueckzahlen.st_ctrl.in.b_stop := FALSE;
			balluff_tag_reader.st_ctrl.in.b_stop := FALSE;
			edit_mfps.st_ctrl.in.b_stop := FALSE;
			axis_transport_wt_achse.st_ctrl.in.b_stop := FALSE;
			(* HALT - nur Achsen *)
			axis_virt_master.st_ctrl.in.b_halt := FALSE;
			axis_bestueckachse.st_ctrl.in.b_halt := FALSE;
			axis_y_achse.st_ctrl.in.b_halt := FALSE;
			axis_z_achse.st_ctrl.in.b_halt := FALSE;
			axis_bandeinzug_achse.st_ctrl.in.b_halt := FALSE;
			axis_transport_wt_achse.st_ctrl.in.b_halt := FALSE;
		END_IF

		IF fb_ton_quitt.Q THEN
			IF (gi16_betriebsart = AUTO OR gi16_betriebsart = TIPPEN) THEN
				fb_state_entry.i16_next_step := INIT;
			END_IF
		END_IF
END_CASE

fb_state_entry(
	i16_next_step:= ,
	i16_pos:= 2,
	s_debugtext:= ,
	E=> ,
	X=> , 
	i16_step=> ,
	i16_last_step=> );


(*Beim Einfädel Meldung zurücksetzen*)
IF	ST_TippTasten.b_einfaedeln_aktiv THEN
	bm_Maschine_in_Gst := FALSE;
END_IF

IF st_config.b_config_fertig THEN
	(* Fehlermeldungen und Betriebsmeldungen ab dem Startindex in die globalen Meldungsarrays schreiben *)
	garr_stoermeldungen[st_config.i16_meld_startindex + 0] := sm_disable_auto_reset;
	garr_stoermeldungen[st_config.i16_meld_startindex + 1] := FALSE;
	garr_stoermeldungen[st_config.i16_meld_startindex + 2] := FALSE;
	garr_stoermeldungen[st_config.i16_meld_startindex + 3] := FALSE;
	garr_stoermeldungen[st_config.i16_meld_startindex + 4] := FALSE;
	garr_stoermeldungen[st_config.i16_meld_startindex + 5] := FALSE;
	garr_stoermeldungen[st_config.i16_meld_startindex + 6] := FALSE;
	garr_stoermeldungen[st_config.i16_meld_startindex + 7] := FALSE;
	garr_stoermeldungen[st_config.i16_meld_startindex + 8] := FALSE;
	garr_stoermeldungen[st_config.i16_meld_startindex + 9] := FALSE;
	garr_stoermeldungen[st_config.i16_meld_startindex + 10] := FALSE;
	garr_stoermeldungen[st_config.i16_meld_startindex + 11] := FALSE;
	garr_stoermeldungen[st_config.i16_meld_startindex + 12] := FALSE;
	garr_stoermeldungen[st_config.i16_meld_startindex + 13] := FALSE;
	garr_stoermeldungen[st_config.i16_meld_startindex + 14] := FALSE;
	garr_stoermeldungen[st_config.i16_meld_startindex + 15] := FALSE;
	garr_stoermeldungen[st_config.i16_meld_startindex + 16] := FALSE;
	garr_stoermeldungen[st_config.i16_meld_startindex + 17] := FALSE;
	garr_stoermeldungen[st_config.i16_meld_startindex + 18] := FALSE;
	garr_stoermeldungen[st_config.i16_meld_startindex + 19] := FALSE;
	
	garr_betriebsmeldungen[st_config.i16_meld_startindex + 0] := bm_Maschine_in_Gst;
	garr_betriebsmeldungen[st_config.i16_meld_startindex + 1] := bm_Check;
	garr_betriebsmeldungen[st_config.i16_meld_startindex + 2] := FALSE;
	garr_betriebsmeldungen[st_config.i16_meld_startindex + 3] := FALSE;
	garr_betriebsmeldungen[st_config.i16_meld_startindex + 4] := FALSE;
	garr_betriebsmeldungen[st_config.i16_meld_startindex + 5] := FALSE;
	garr_betriebsmeldungen[st_config.i16_meld_startindex + 6] := FALSE;
	garr_betriebsmeldungen[st_config.i16_meld_startindex + 7] := FALSE;
	garr_betriebsmeldungen[st_config.i16_meld_startindex + 8] := FALSE;
	garr_betriebsmeldungen[st_config.i16_meld_startindex + 9] := FALSE;
	garr_betriebsmeldungen[st_config.i16_meld_startindex + 10] := FALSE;
	garr_betriebsmeldungen[st_config.i16_meld_startindex + 11] := FALSE;
	garr_betriebsmeldungen[st_config.i16_meld_startindex + 12] := FALSE;
	garr_betriebsmeldungen[st_config.i16_meld_startindex + 13] := FALSE;
	garr_betriebsmeldungen[st_config.i16_meld_startindex + 14] := FALSE;
	garr_betriebsmeldungen[st_config.i16_meld_startindex + 15] := FALSE;
	garr_betriebsmeldungen[st_config.i16_meld_startindex + 16] := FALSE;
	garr_betriebsmeldungen[st_config.i16_meld_startindex + 17] := FALSE;
	garr_betriebsmeldungen[st_config.i16_meld_startindex + 18] := FALSE;
	garr_betriebsmeldungen[st_config.i16_meld_startindex + 19] := FALSE;
END_IF
END_PROGRAM

(* POU Maschine1720/ST_Stoerungen_Quitt_1720, ST *)
PROGRAM ST_Stoerungen_Quitt_1720
VAR_INPUT
	st_config					: struct_config;
	st_ctrl_in					: struct_ctrl_in;
END_VAR
VAR_IN_OUT
	st_visu					: struct_visu;
	st_visu_hinten				: struct_visu_hinten;
END_VAR
VAR_OUTPUT
	st_ctrl_out				: struct_ctrl_out;
	b_lampe_stoerung		: BOOL;
	b_lampe_produktion		: BOOL;
END_VAR
VAR
	fb_ton_quitt				: TON;
	fb_r_trig_quittieren			: R_TRIG;
	b_Merker_quitt			: BOOL:=FALSE;
	fb_ton_wz				: TON;

	fb_state_entry				: ST_StateEntry;

	fb_blinker				: ST_Blinker;

	bm_Maschine_in_Gst		: BOOL := FALSE;
	bm_Check		: BOOL := FALSE;
	sm_disable_auto_reset	: BOOL := FALSE;
END_VAR
(* Zeiten *)
fb_ton_quitt(IN:= , PT:= t#300ms, Q=> , ET=> );

(* Flanken *)
fb_r_trig_quittieren(CLK:= (st_visu.b_quittieren OR st_visu_hinten.out.b_quittieren) AND gi16_betriebsart <> HAND, Q=> );

(* Blinker *)
fb_blinker(
	b_start:= TRUE,
	t_taktzeit_on:=t#500ms,
	t_taktzeit_off:=t#500ms,
	b_blinker_out=> );

(* Lampen *)
b_lampe_stoerung := gi16_maschinenstatusinfo = KEIN_STATUS OR gi16_maschinenstatusinfo = STATUS_FEHLER;

b_lampe_produktion := (fb_blinker.b_blinker_out AND
					(gi16_maschinenstatusinfo = STATUS_FEHLER_QUITTIERT OR
					gi16_maschinenstatusinfo = STATUS_BETRIEBSBEREIT)) OR
					gi16_maschinenstatusinfo = STATUS_MASCHINE_ARBEITET;

bm_Check:=(
	CheckBounds_ErrCnt+
	CheckByteZeroDiv_ErrCnt+
	CheckDWordZeroDiv_ErrCnt+
	CheckRealZeroDiv_ErrCnt+
	CheckWordZeroDiv_ErrCnt+
	CheckRangeSigned_ErrCnt+
	CheckRangeUnsigned_ErrCnt) > 0 ;

(* Toplevel *)
(* Hier nur Abschaltungen welche zu sofortigem Stop führen müssen *)
IF fb_state_entry.i16_step < FEHLER AND
	(axis_virt_master.st_ctrl.out.b_fehler OR
	axis_bestueckachse.st_ctrl.out.b_fehler OR
	axis_z_achse.st_ctrl.out.b_fehler OR
	bandeinzug_kontroller.st_ctrl.out.b_fehler OR
	bandspruehoeler.st_ctrl.out.b_fehler OR
	wkz_absicherung.st_ctrl.out.b_fehler OR
	wt_transport_kontroller.st_ctrl.out.b_fehler OR
(*	hublift_links.st_ctrl.out.b_fehler OR
	hublift_rechts.st_ctrl.out.b_fehler OR*)
	balluff_tag_reader.st_ctrl.out.b_fehler OR
	haspel_kontroller.st_ctrl.out.b_fehler OR
	bbgen.st_ctrl.out.b_fehler OR
	wartung.st_ctrl.out.b_fehler OR
	betriebsfreigaben.st_ctrl.out.b_fehler OR
	safety.st_ctrl.out.b_fehler OR
	edit_mfps.st_ctrl.out.b_fehler OR
	Lesen_Schreiben_Tag.st_ctrl.out.b_fehler OR
	Service.st_ctrl.out.b_fehler)
	THEN
		fb_state_entry.i16_next_step := FEHLER;
END_IF

(* Prüfe ob BA = Hand -> Stoppe Abläufe *)
IF  fb_state_entry.i16_step > INIT  AND fb_state_entry.i16_step < FEHLER  AND gi16_betriebsart = HAND THEN
	fb_state_entry.i16_next_step := FEHLER;
END_IF

(* ======================================Schrittkette======================================== *)
fb_state_entry(
	i16_next_step:= ,
	i16_pos:= 1,
	s_debugtext:= ,
	E=> ,
	X=> ,
	i16_step=> ,
	i16_last_step=> );

CASE fb_state_entry.i16_step OF
(*=======================================================*)
	INIT_OBJ:
		IF st_config.b_config_fertig THEN
			fb_state_entry.i16_next_step := FEHLER;
		END_IF

(*=======================================================*)
	INIT:
		IF fb_state_entry.E THEN
			gi16_maschinenstatusinfo := STATUS_FEHLER_QUITTIERT;

			fb_ton_quitt.IN := FALSE;
			UPS.st_ctrl.in.b_quitt := FALSE;
			betriebsfreigaben.st_ctrl.in.b_quitt := FALSE;
			bandeinzug_kontroller.st_ctrl.in.b_quitt := FALSE;
			axis_virt_master.st_ctrl.in.b_quitt := FALSE;
			axis_bestueckachse.st_ctrl.in.b_quitt := FALSE;
			axis_z_achse.st_ctrl.in.b_quitt := FALSE;
			bandspruehoeler.st_ctrl.in.b_quitt := FALSE;
			haspel_kontroller.st_ctrl.in.b_quitt := FALSE;
			hublift_links.st_ctrl.in.b_quitt := FALSE;
			hublift_rechts.st_ctrl.in.b_quitt := FALSE;
			wt_transport_kontroller.st_ctrl.in.b_quitt := FALSE;
			wkz_absicherung.st_ctrl.in.b_quitt := FALSE;
			stueckzahlen.st_ctrl.in.b_quitt := FALSE;
			balluff_tag_reader.st_ctrl.in.b_quitt := FALSE;
			bbgen.st_ctrl.in.b_quitt := FALSE;
			wartung.st_ctrl.in.b_quitt := FALSE;
			safety.st_ctrl.in.b_quitt := FALSE;
			edit_mfps.st_ctrl.in.b_quitt := FALSE;
			routing_backpanel.st_ctrl.in.b_quitt := FALSE;
			routing_nachbarpc.st_ctrl.in.b_quitt := FALSE;
			bm_Maschine_in_Gst := FALSE;
			Lesen_Schreiben_Tag.st_ctrl.in.b_quitt :=FALSE;
			Service.st_ctrl.in.b_quitt :=FALSE;
			ST_TippTasten.b_initialisierungsphase := TRUE;
			sm_disable_auto_reset := FALSE;
		END_IF

		(*-----------------------Weiterschaltbedingungen----------------------------*)
		IF safety.st_ctrl.out.b_bereit THEN
			fb_state_entry.i16_next_step := 11;
		END_IF

(*=======================================================*)
	11:
		IF fb_state_entry.E THEN
			axis_virt_master.st_ctrl.in.b_preinit := TRUE;
		END_IF

		(*-----------------------Weiterschaltbedingungen----------------------------*)
		IF axis_virt_master.st_ctrl.out.b_prebereit  THEN
			axis_virt_master.st_ctrl.in.b_preinit := FALSE;
			fb_state_entry.i16_next_step := 12;
		END_IF

(*=======================================================*)
	12:
		IF fb_state_entry.E THEN
			axis_z_achse.st_ctrl.in.b_preinit := TRUE;
		END_IF

		(*-----------------------Weiterschaltbedingungen----------------------------*)
		IF axis_z_achse.st_ctrl.out.b_prebereit  THEN
			axis_z_achse.st_ctrl.in.b_preinit := FALSE;
			fb_state_entry.i16_next_step := 14;
		END_IF

(*=======================================================*)
	14:
		IF fb_state_entry.E THEN
			axis_bestueckachse.st_ctrl.in.b_preinit := TRUE;
		END_IF

		(*-----------------------Weiterschaltbedingungen----------------------------*)
		IF axis_bestueckachse.st_ctrl.out.b_prebereit THEN
			axis_bestueckachse.st_ctrl.in.b_preinit := FALSE;
			fb_state_entry.i16_next_step := 16;
		END_IF

(*=======================================================*)
	16:
		(*Wenn die Bestückachse nicht in einem bestimmten Bereich steht, dann muss sie von Hand
		    freigefahren werden. Außer es ist die Nocke auf 0,0 gestellt*)
		IF	gst_datensatz.st_wkz.nockenschaltwerk_bestueckachse.arr_nocken[SP_DISABLE_AUTO_RESET].r_cam_begin = 0 AND
			gst_datensatz.st_wkz.nockenschaltwerk_bestueckachse.arr_nocken[SP_DISABLE_AUTO_RESET].r_cam_end = 0 THEN
				fb_state_entry.i16_next_step := 20;
		ELSE
			IF gst_datensatz.st_wkz.nockenschaltwerk_bestueckachse.arr_nocken[SP_DISABLE_AUTO_RESET].r_cam_begin > gst_datensatz.st_wkz.nockenschaltwerk_bestueckachse.arr_nocken[SP_DISABLE_AUTO_RESET].r_cam_end THEN
				IF bestueckachse.NcToPlc.ModuloActPos > gst_datensatz.st_wkz.nockenschaltwerk_bestueckachse.arr_nocken[SP_DISABLE_AUTO_RESET].r_cam_begin OR
					bestueckachse.NcToPlc.ModuloActPos < gst_datensatz.st_wkz.nockenschaltwerk_bestueckachse.arr_nocken[SP_DISABLE_AUTO_RESET].r_cam_end THEN
					sm_disable_auto_reset := TRUE;
					fb_state_entry.i16_next_step := FEHLER;
				ELSE
					fb_state_entry.i16_next_step := 20;
				END_IF
			ELSE
				IF bestueckachse.NcToPlc.ModuloActPos > gst_datensatz.st_wkz.nockenschaltwerk_bestueckachse.arr_nocken[SP_DISABLE_AUTO_RESET].r_cam_begin AND
					bestueckachse.NcToPlc.ModuloActPos < gst_datensatz.st_wkz.nockenschaltwerk_bestueckachse.arr_nocken[SP_DISABLE_AUTO_RESET].r_cam_end THEN
					sm_disable_auto_reset := TRUE;
					fb_state_entry.i16_next_step := FEHLER;
				ELSE
					fb_state_entry.i16_next_step := 20;
				END_IF
			END_IF
		END_IF

(*=======================================================*)
	20:
		IF fb_state_entry.E THEN
			haspel_kontroller.st_ctrl.in.b_init := TRUE;
			bandspruehoeler.st_ctrl.in.b_init := TRUE;
			wkz_absicherung.st_ctrl.in.b_init := TRUE;
			stueckzahlen.st_ctrl.in.b_init := TRUE;
			(*balluff_tag_reader.st_ctrl.in.b_init := TRUE;*)
			edit_mfps.st_ctrl.in.b_init := TRUE;
		END_IF

		(*-----------------------Weiterschaltbedingungen----------------------------*)
		IF 	haspel_kontroller.st_ctrl.out.b_bereit  AND
			bandspruehoeler.st_ctrl.out.b_bereit  AND
			wkz_absicherung.st_ctrl.out.b_bereit AND
			balluff_tag_reader.st_ctrl.out.b_bereit AND
			edit_mfps.st_ctrl.out.b_bereit
			THEN
				haspel_kontroller.st_ctrl.in.b_init := FALSE;
				bandspruehoeler.st_ctrl.in.b_init := FALSE;
				wkz_absicherung.st_ctrl.in.b_init := FALSE;
				stueckzahlen.st_ctrl.in.b_init := FALSE;
				(*balluff_tag_reader.st_ctrl.in.b_init := FALSE;*)
				edit_mfps.st_ctrl.in.b_init := FALSE;
				fb_state_entry.i16_next_step := 30;
		END_IF

(*=======================================================*)
	30:
		IF fb_state_entry.E THEN
			bandeinzug_kontroller.st_ctrl.in.b_init := TRUE;
		END_IF

		(*-----------------------Weiterschaltbedingungen----------------------------*)
		IF bandeinzug_kontroller.st_ctrl.out.b_bereit THEN
			bandeinzug_kontroller.st_ctrl.in.b_init := FALSE;
			fb_state_entry.i16_next_step := 40;
		END_IF

(*=======================================================*)
	40:
		IF fb_state_entry.E THEN
			axis_bestueckachse.st_ctrl.in.b_init := TRUE;
		END_IF

		(*-----------------------Weiterschaltbedingungen----------------------------*)
		IF axis_bestueckachse.st_ctrl.out.b_bereit  THEN
			axis_bestueckachse.st_ctrl.in.b_init := FALSE;
			fb_state_entry.i16_next_step := 50;
		END_IF

(*=======================================================*)
	50:
		IF fb_state_entry.E THEN
			axis_z_achse.st_ctrl.in.b_init := TRUE;
		END_IF

		(*-----------------------Weiterschaltbedingungen----------------------------*)
		IF axis_z_achse.st_ctrl.out.b_bereit THEN
			axis_z_achse.st_ctrl.in.b_init := FALSE;
			fb_state_entry.i16_next_step := 60;
		END_IF

(*=======================================================*)
	60:
		IF fb_state_entry.E THEN
			axis_virt_master.st_ctrl.in.b_init := TRUE;
		END_IF

		(*-----------------------Weiterschaltbedingungen----------------------------*)
		IF axis_virt_master.st_ctrl.out.b_bereit  THEN
			axis_virt_master.st_ctrl.in.b_init := FALSE;
			fb_state_entry.i16_next_step := 70;
		END_IF

(*=======================================================*)
	70:
		IF fb_state_entry.E THEN
			hublift_links.st_ctrl.in.b_init := TRUE;
			hublift_rechts.st_ctrl.in.b_init := TRUE;
			wt_transport_kontroller.st_ctrl.in.b_init := TRUE;
		END_IF

		(*-----------------------Weiterschaltbedingungen----------------------------*)
		IF hublift_links.st_ctrl.out.b_bereit AND hublift_rechts.st_ctrl.out.b_bereit AND wt_transport_kontroller.st_ctrl.out.b_bereit THEN
			hublift_links.st_ctrl.in.b_init := FALSE;
			hublift_rechts.st_ctrl.in.b_init := FALSE;
			wt_transport_kontroller.st_ctrl.in.b_init := FALSE;
			fb_state_entry.i16_next_step := BEREIT;
		END_IF

(*=======================================================*)
	BEREIT:
		IF fb_state_entry.E THEN
			ST_TippTasten.b_initialisierungsphase  := FALSE;

			(* Setze Maschinenstatus *)
			bm_Maschine_in_Gst := TRUE;
		END_IF

		(*Beim Einfädeln muss der Status geändert werden, damit nicht
		ständig neue Maschinendaten erzeugt werden*)
		IF ST_TippTasten.b_einfaedeln_aktiv THEN
			gi16_maschinenstatusinfo := STATUS_MASCHINE_ARBEITET;
		ELSE
			gi16_maschinenstatusinfo := STATUS_BETRIEBSBEREIT;
		END_IF

		(*-----------------------Weiterschaltbedingungen----------------------------*)
		IF NOT wt_transport_kontroller.st_ctrl.out.b_fertig THEN
			bm_Maschine_in_Gst := FALSE;
			fb_state_entry.i16_next_step := 110;
		END_IF

(*=======================================================*)
	110: (* Produktion *)
		IF fb_state_entry.E THEN
			gi16_maschinenstatusinfo := STATUS_MASCHINE_ARBEITET;
		END_IF

		(*-----------------------Weiterschaltbedingungen----------------------------*)
		IF wt_transport_kontroller.st_ctrl.out.b_fertig THEN
			fb_state_entry.i16_next_step := BEREIT;
		END_IF

(*=======================================================*)
	FEHLER:
		IF fb_state_entry.E THEN
			gi16_maschinenstatusinfo := STATUS_FEHLER;
			bm_Maschine_in_Gst := FALSE;
			ST_TippTasten.b_initialisierungsphase  := FALSE;
			fb_ton_quitt.IN := FALSE;
			fb_ton_wz.IN:=FALSE;
			s_alte_artikelnummer := '';

			(* Schlecht Stueckzahl erhöhen *)
			IF fb_state_entry.i16_last_step = 110 THEN
				stueckzahlen.st_ctrl.in.b_schlechtteil_produziert := TRUE;
			END_IF

			UPS.st_ctrl.in.b_quitt := FALSE;
			betriebsfreigaben.st_ctrl.in.b_quitt := FALSE;
			bandeinzug_kontroller.st_ctrl.in.b_quitt := FALSE;
			axis_virt_master.st_ctrl.in.b_quitt := FALSE;
			axis_bestueckachse.st_ctrl.in.b_quitt := FALSE;
			axis_z_achse.st_ctrl.in.b_quitt := FALSE;
			bandspruehoeler.st_ctrl.in.b_quitt := FALSE;
			haspel_kontroller.st_ctrl.in.b_quitt := FALSE;
			hublift_links.st_ctrl.in.b_quitt := FALSE;
			hublift_rechts.st_ctrl.in.b_quitt := FALSE;
			wt_transport_kontroller.st_ctrl.in.b_quitt := FALSE;
			wkz_absicherung.st_ctrl.in.b_quitt := FALSE;
			stueckzahlen.st_ctrl.in.b_quitt := FALSE;
			balluff_tag_reader.st_ctrl.in.b_quitt := FALSE;
			bbgen.st_ctrl.in.b_quitt := FALSE;
			wartung.st_ctrl.in.b_quitt := FALSE;
			safety.st_ctrl.in.b_quitt := FALSE;
			edit_mfps.st_ctrl.in.b_quitt := FALSE;
			routing_backpanel.st_ctrl.in.b_quitt := FALSE;
			routing_nachbarpc.st_ctrl.in.b_quitt := FALSE;
			Lesen_Schreiben_Tag.st_ctrl.in.b_quitt := FALSE;
			Service.st_ctrl.in.b_quitt := FALSE;

			axis_virt_master.st_ctrl.in.b_preinit := FALSE;
			axis_bestueckachse.st_ctrl.in.b_preinit := FALSE;
			axis_z_achse.st_ctrl.in.b_preinit := FALSE;

			bandeinzug_kontroller.st_ctrl.in.b_init := FALSE;
			axis_virt_master.st_ctrl.in.b_init := FALSE;
			axis_bestueckachse.st_ctrl.in.b_init := FALSE;
			axis_z_achse.st_ctrl.in.b_init := FALSE;
			bandspruehoeler.st_ctrl.in.b_init := FALSE;
			haspel_kontroller.st_ctrl.in.b_init := FALSE;
			hublift_links.st_ctrl.in.b_init := FALSE;
			hublift_rechts.st_ctrl.in.b_init := FALSE;
			wt_transport_kontroller.st_ctrl.in.b_init := FALSE;
			wkz_absicherung.st_ctrl.in.b_init := FALSE;
			stueckzahlen.st_ctrl.in.b_init := FALSE;
			balluff_tag_reader.st_ctrl.in.b_init := FALSE;
			edit_mfps.st_ctrl.in.b_init := FALSE;
		END_IF

		(* Fehlerhandling: was soll bei welchem Fehler passieren? *)
		IF 	NOT fb_ton_quitt.IN THEN
			(* Stoppe/Halte Komponenten an *)
			bandeinzug_kontroller.st_ctrl.in.b_stop := TRUE;
			bandspruehoeler.st_ctrl.in.b_stop := TRUE;
			(*haspel_kontroller.st_ctrl.in.b_stop := TRUE;*)
			hublift_links.st_ctrl.in.b_stop := TRUE;
			hublift_rechts.st_ctrl.in.b_stop := TRUE;
			wt_transport_kontroller.st_ctrl.in.b_stop := TRUE;
			stueckzahlen.st_ctrl.in.b_stop := TRUE;
			balluff_tag_reader.st_ctrl.in.b_stop := TRUE;
			edit_mfps.st_ctrl.in.b_stop := TRUE;

			(* Diese Fehler führt zum "Stop" in der Maschine *)
			IF safety.st_ctrl.out.b_fehler THEN
				axis_virt_master.st_ctrl.in.b_stop := TRUE;
				axis_bestueckachse.st_ctrl.in.b_stop := TRUE;
				axis_z_achse.st_ctrl.in.b_stop := TRUE;
				axis_virt_master.st_ctrl.in.b_halt := FALSE;
				axis_bestueckachse.st_ctrl.in.b_halt := FALSE;
				axis_z_achse.st_ctrl.in.b_halt := FALSE;
			ELSE
				axis_virt_master.st_ctrl.in.b_halt := TRUE;
				axis_bestueckachse.st_ctrl.in.b_halt := TRUE;
				axis_z_achse.st_ctrl.in.b_halt := TRUE;
				axis_virt_master.st_ctrl.in.b_stop := FALSE;
				axis_bestueckachse.st_ctrl.in.b_stop := FALSE;
				axis_z_achse.st_ctrl.in.b_stop := FALSE;
			END_IF
		END_IF

		(*-----------------------Weiterschaltbedingungen----------------------------*)
		IF 	fb_r_trig_quittieren.Q THEN
			fb_ton_wz.IN:=TRUE;
			b_Merker_quitt:=TRUE;
		END_IF
		IF 	(b_Merker_quitt AND ST_Betriebsfreigaben.e_druckwaechter) OR
			fb_ton_wz.Q THEN
			fb_ton_wz.IN:=FALSE;
			b_Merker_quitt:=FALSE;
			fb_ton_quitt.IN := TRUE;
			(* QUITT *)
			UPS.st_ctrl.in.b_quitt := TRUE;
			betriebsfreigaben.st_ctrl.in.b_quitt := TRUE;
			bandeinzug_kontroller.st_ctrl.in.b_quitt := TRUE;
			axis_virt_master.st_ctrl.in.b_quitt := TRUE;
			axis_bestueckachse.st_ctrl.in.b_quitt := TRUE;
			axis_z_achse.st_ctrl.in.b_quitt := TRUE;
			bandspruehoeler.st_ctrl.in.b_quitt := TRUE;
			haspel_kontroller.st_ctrl.in.b_quitt := TRUE;
			hublift_links.st_ctrl.in.b_quitt := TRUE;
			hublift_rechts.st_ctrl.in.b_quitt := TRUE;
			wt_transport_kontroller.st_ctrl.in.b_quitt := TRUE;
			wkz_absicherung.st_ctrl.in.b_quitt := TRUE;
			stueckzahlen.st_ctrl.in.b_quitt := TRUE;
			balluff_tag_reader.st_ctrl.in.b_quitt := TRUE;
			bbgen.st_ctrl.in.b_quitt := TRUE;
			wartung.st_ctrl.in.b_quitt := TRUE;
			safety.st_ctrl.in.b_quitt := TRUE;
			edit_mfps.st_ctrl.in.b_quitt := TRUE;
			routing_backpanel.st_ctrl.in.b_quitt := TRUE;
			routing_nachbarpc.st_ctrl.in.b_quitt := TRUE;
			Lesen_Schreiben_Tag.st_ctrl.in.b_quitt := TRUE;
			Service.st_ctrl.in.b_quitt := TRUE;
			(* STOP *)
			bandeinzug_kontroller.st_ctrl.in.b_stop := FALSE;
			axis_virt_master.st_ctrl.in.b_stop := FALSE;
			axis_bestueckachse.st_ctrl.in.b_stop := FALSE;
			axis_z_achse.st_ctrl.in.b_stop := FALSE;
			bandspruehoeler.st_ctrl.in.b_stop := FALSE;
			haspel_kontroller.st_ctrl.in.b_stop := FALSE;
			hublift_links.st_ctrl.in.b_stop := FALSE;
			hublift_rechts.st_ctrl.in.b_stop := FALSE;
			wt_transport_kontroller.st_ctrl.in.b_stop := FALSE;
			wkz_absicherung.st_ctrl.in.b_stop := FALSE;
			stueckzahlen.st_ctrl.in.b_stop := FALSE;
			balluff_tag_reader.st_ctrl.in.b_stop := FALSE;
			edit_mfps.st_ctrl.in.b_stop := FALSE;
			(* HALT - nur Achsen *)
			axis_virt_master.st_ctrl.in.b_halt := FALSE;
			axis_bestueckachse.st_ctrl.in.b_halt := FALSE;
			axis_z_achse.st_ctrl.in.b_halt := FALSE;
		END_IF

		IF fb_ton_quitt.Q THEN
			IF (gi16_betriebsart = AUTO OR gi16_betriebsart = TIPPEN) THEN
				fb_state_entry.i16_next_step := INIT;
			END_IF
		END_IF
END_CASE

fb_state_entry(
	i16_next_step:= ,
	i16_pos:= 2,
	s_debugtext:= ,
	E=> ,
	X=> , 
	i16_step=> ,
	i16_last_step=> );

IF st_config.b_config_fertig THEN
	(* Fehlermeldungen und Betriebsmeldungen ab dem Startindex in die globalen Meldungsarrays schreiben *)
	garr_stoermeldungen[st_config.i16_meld_startindex + 0] := sm_disable_auto_reset;
	garr_stoermeldungen[st_config.i16_meld_startindex + 1] := FALSE;
	garr_stoermeldungen[st_config.i16_meld_startindex + 2] := FALSE;
	garr_stoermeldungen[st_config.i16_meld_startindex + 3] := FALSE;
	garr_stoermeldungen[st_config.i16_meld_startindex + 4] := FALSE;
	garr_stoermeldungen[st_config.i16_meld_startindex + 5] := FALSE;
	garr_stoermeldungen[st_config.i16_meld_startindex + 6] := FALSE;
	garr_stoermeldungen[st_config.i16_meld_startindex + 7] := FALSE;
	garr_stoermeldungen[st_config.i16_meld_startindex + 8] := FALSE;
	garr_stoermeldungen[st_config.i16_meld_startindex + 9] := FALSE;
	garr_stoermeldungen[st_config.i16_meld_startindex + 10] := FALSE;
	garr_stoermeldungen[st_config.i16_meld_startindex + 11] := FALSE;
	garr_stoermeldungen[st_config.i16_meld_startindex + 12] := FALSE;
	garr_stoermeldungen[st_config.i16_meld_startindex + 13] := FALSE;
	garr_stoermeldungen[st_config.i16_meld_startindex + 14] := FALSE;
	garr_stoermeldungen[st_config.i16_meld_startindex + 15] := FALSE;
	garr_stoermeldungen[st_config.i16_meld_startindex + 16] := FALSE;
	garr_stoermeldungen[st_config.i16_meld_startindex + 17] := FALSE;
	garr_stoermeldungen[st_config.i16_meld_startindex + 18] := FALSE;
	garr_stoermeldungen[st_config.i16_meld_startindex + 19] := FALSE;
	
	garr_betriebsmeldungen[st_config.i16_meld_startindex + 0] := bm_Maschine_in_Gst;
	garr_betriebsmeldungen[st_config.i16_meld_startindex + 1] := bm_Check;
	garr_betriebsmeldungen[st_config.i16_meld_startindex + 2] := FALSE;
	garr_betriebsmeldungen[st_config.i16_meld_startindex + 3] := FALSE;
	garr_betriebsmeldungen[st_config.i16_meld_startindex + 4] := FALSE;
	garr_betriebsmeldungen[st_config.i16_meld_startindex + 5] := FALSE;
	garr_betriebsmeldungen[st_config.i16_meld_startindex + 6] := FALSE;
	garr_betriebsmeldungen[st_config.i16_meld_startindex + 7] := FALSE;
	garr_betriebsmeldungen[st_config.i16_meld_startindex + 8] := FALSE;
	garr_betriebsmeldungen[st_config.i16_meld_startindex + 9] := FALSE;
	garr_betriebsmeldungen[st_config.i16_meld_startindex + 10] := FALSE;
	garr_betriebsmeldungen[st_config.i16_meld_startindex + 11] := FALSE;
	garr_betriebsmeldungen[st_config.i16_meld_startindex + 12] := FALSE;
	garr_betriebsmeldungen[st_config.i16_meld_startindex + 13] := FALSE;
	garr_betriebsmeldungen[st_config.i16_meld_startindex + 14] := FALSE;
	garr_betriebsmeldungen[st_config.i16_meld_startindex + 15] := FALSE;
	garr_betriebsmeldungen[st_config.i16_meld_startindex + 16] := FALSE;
	garr_betriebsmeldungen[st_config.i16_meld_startindex + 17] := FALSE;
	garr_betriebsmeldungen[st_config.i16_meld_startindex + 18] := FALSE;
	garr_betriebsmeldungen[st_config.i16_meld_startindex + 19] := FALSE;
END_IF
END_PROGRAM

(* POU Maschine1720/ST_AbfallBlasluft, ST *)
PROGRAM ST_AbfallBlasluft
VAR_INPUT
	b_wkz_blasluft_aktiv	: BOOL;
END_VAR
VAR
	a_AbfallBlasluft		AT %Q* : BOOL;
	fb_rtrig_nocke		: R_TRIG;
	fb_tof_blaszeit		: TOF;
	b_blasluft_aktiv		: BOOL := FALSE;
END_VAR
fb_rtrig_nocke (CLK:= (bestueckachse.NcToPlc.ModuloActPos > 170 AND bestueckachse.NcToPlc.ModuloActPos < 190), Q=> );

IF b_wkz_blasluft_aktiv THEN
	fb_tof_blaszeit (IN:=fb_rtrig_nocke.Q , PT:= t#200ms, Q=> a_AbfallBlasluft, ET=> );
END_IF
END_PROGRAM

(* POU Rasterfolie/ST_Rafl_Stoerungen_Quitt, ST *)
PROGRAM ST_Rafl_Stoerungen_Quitt
VAR_INPUT
	st_config						: struct_config;
	st_ctrl_in						: struct_ctrl_in;
END_VAR
VAR_IN_OUT
	st_visu						: struct_visu;
	st_visu_hinten					: struct_visu_hinten;
END_VAR
VAR_OUTPUT
	st_ctrl_out					: struct_ctrl_out;
	b_lampe_stoerung			: BOOL;
	b_lampe_produktion			: BOOL;
END_VAR
VAR
	fb_ton_quitt					: TON;
	fb_ton_wz				: TON;
	fb_r_trig_quittieren				: R_TRIG;
	fb_state_entry					: ST_StateEntry;

	fb_blinker					: ST_Blinker;
	b_Merker_quitt			: BOOL:=FALSE;
	bm_Maschine_in_Gst			: BOOL := FALSE;
END_VAR
(* Zeiten *)
fb_ton_quitt(IN:= , PT:= t#150ms, Q=> , ET=> );
fb_ton_wz(IN:= , PT:= t#3000ms, Q=> , ET=> );

(* Flanken *)
fb_r_trig_quittieren(CLK:= (st_visu.b_quittieren OR st_visu_hinten.out.b_quittieren) AND gi16_betriebsart <> HAND, Q=> );

(* Blinker *)
fb_blinker(
	b_start:= TRUE,
	t_taktzeit_on:=t#500ms,
	t_taktzeit_off:=t#500ms,
	b_blinker_out=> );

(* Lampen *)
b_lampe_stoerung := gi16_maschinenstatusinfo = KEIN_STATUS OR gi16_maschinenstatusinfo = STATUS_FEHLER;

b_lampe_produktion := (fb_blinker.b_blinker_out AND
					(gi16_maschinenstatusinfo = STATUS_FEHLER_QUITTIERT OR
					gi16_maschinenstatusinfo = STATUS_BETRIEBSBEREIT)) OR
					gi16_maschinenstatusinfo = STATUS_MASCHINE_ARBEITET;

(* Toplevel *)
(* Hier nur Abschaltungen welche zu sofortigem Stop führen müssen *)
IF fb_state_entry.i16_step < FEHLER AND
	(axis_virt_master.st_ctrl.out.b_fehler OR
	axis_bestueckachse.st_ctrl.out.b_fehler OR
	axis_z_achse.st_ctrl.out.b_fehler OR
	axis_y_achse.st_ctrl.out.b_fehler OR
	ST_TouchProbe.st_ctrl_out.b_fehler OR
	haspel_kontroller.st_ctrl.out.b_fehler OR
	rasterfolieneinzug.st_ctrl.out.b_fehler OR
	rasterfolienmontage.st_ctrl.out.b_fehler OR
	wt_transport_kontroller.st_ctrl.out.b_fehler OR
	balluff_tag_reader.st_ctrl.out.b_fehler OR
	bbgen.st_ctrl.out.b_fehler OR
	betriebsfreigaben.st_ctrl.out.b_fehler OR
	safety.st_ctrl.out.b_fehler OR
	edit_mfps.st_ctrl.out.b_fehler OR
	Lesen_Schreiben_Tag.st_ctrl.out.b_fehler OR
	Service.st_ctrl.out.b_fehler)
	THEN
		fb_state_entry.i16_next_step := FEHLER;
END_IF

(* Prüfe ob BA = Hand -> Stoppe Abläufe *)
IF  fb_state_entry.i16_step > INIT  AND fb_state_entry.i16_step < FEHLER  AND gi16_betriebsart = HAND THEN
	fb_state_entry.i16_next_step := FEHLER;
END_IF

(* ======================================Schrittkette======================================== *)
fb_state_entry(
	i16_next_step:= ,
	i16_pos:= 1,
	s_debugtext:= ,
	E=> ,
	X=> ,
	i16_step=> ,
	i16_last_step=> );

CASE fb_state_entry.i16_step OF
(*=======================================================*)
	INIT_OBJ:
		IF st_config.b_config_fertig THEN
			fb_state_entry.i16_next_step := FEHLER;
		END_IF

(*=======================================================*)
	INIT:
		IF fb_state_entry.E THEN
			gi16_maschinenstatusinfo := STATUS_FEHLER_QUITTIERT;
			fb_ton_quitt.IN := FALSE;
			betriebsfreigaben.st_ctrl.in.b_quitt := FALSE;
			safety.st_ctrl.in.b_quitt := FALSE;
			rasterfolienmontage.st_ctrl.in.b_quitt := FALSE;
			rasterfolieneinzug.st_ctrl.in.b_quitt := FALSE;
			axis_virt_master.st_ctrl.in.b_quitt := FALSE;
			axis_bestueckachse.st_ctrl.in.b_quitt := FALSE;
			axis_y_achse.st_ctrl.in.b_quitt := FALSE;
			axis_z_achse.st_ctrl.in.b_quitt := FALSE;
			ST_TouchProbe.st_ctrl_in.b_quitt := FALSE;
			hublift_links.st_ctrl.in.b_quitt := FALSE;
			hublift_rechts.st_ctrl.in.b_quitt := FALSE;
			stueckzahlen.st_ctrl.in.b_quitt := FALSE;
			wt_transport_kontroller.st_ctrl.in.b_quitt := FALSE;
			balluff_tag_reader.st_ctrl.in.b_quitt := FALSE;
			bbgen.st_ctrl.in.b_quitt := FALSE;
			edit_mfps.st_ctrl.in.b_quitt := FALSE;
			routing_backpanel.st_ctrl.in.b_quitt := FALSE;
			routing_nachbarpc.st_ctrl.in.b_quitt := FALSE;
			bm_Maschine_in_Gst := FALSE;
			Lesen_Schreiben_Tag.st_ctrl.in.b_quitt := FALSE;
			Service.st_ctrl.in.b_quitt := FALSE;
			ST_TippTasten.b_initialisierungsphase  := TRUE;
			haspel_kontroller.st_ctrl.in.b_quitt := FALSE;
		END_IF

		(*-----------------------Weiterschaltbedingungen----------------------------*)
		IF safety.st_ctrl.out.b_bereit THEN
			fb_state_entry.i16_next_step := 11;
		END_IF

(*=======================================================*)
	11:
		IF fb_state_entry.E THEN
			axis_virt_master.st_ctrl.in.b_preinit := TRUE;
		END_IF

		(*-----------------------Weiterschaltbedingungen----------------------------*)
		IF axis_virt_master.st_ctrl.out.b_prebereit  THEN
			axis_virt_master.st_ctrl.in.b_preinit := FALSE;
			fb_state_entry.i16_next_step := 12;
		END_IF

(*=======================================================*)
	12:
		IF fb_state_entry.E THEN
			axis_z_achse.st_ctrl.in.b_preinit := TRUE;
		END_IF

		(*-----------------------Weiterschaltbedingungen----------------------------*)
		IF axis_z_achse.st_ctrl.out.b_prebereit  THEN
			axis_z_achse.st_ctrl.in.b_preinit := FALSE;
			fb_state_entry.i16_next_step := 14;
		END_IF

(*=======================================================*)
	14:
		IF fb_state_entry.E THEN
			axis_y_achse.st_ctrl.in.b_preinit := TRUE;
		END_IF

		(*-----------------------Weiterschaltbedingungen----------------------------*)
		IF axis_y_achse.st_ctrl.out.b_prebereit  THEN
			axis_y_achse.st_ctrl.in.b_preinit := FALSE;
			fb_state_entry.i16_next_step := 16;
		END_IF

(*=======================================================*)
	16:
		IF fb_state_entry.E THEN
			axis_bestueckachse.st_ctrl.in.b_preinit := TRUE;
		END_IF

		(*-----------------------Weiterschaltbedingungen----------------------------*)
		IF axis_bestueckachse.st_ctrl.out.b_prebereit THEN
			axis_bestueckachse.st_ctrl.in.b_preinit := FALSE;
			fb_state_entry.i16_next_step := 20;
		END_IF

(*=======================================================*)
	20:
		IF fb_state_entry.E THEN
			haspel_kontroller.st_ctrl.in.b_init := TRUE;
			stueckzahlen.st_ctrl.in.b_init := TRUE;
			balluff_tag_reader.st_ctrl.in.b_init := TRUE;
			rasterfolienmontage.st_ctrl.in.b_init := TRUE;
			edit_mfps.st_ctrl.in.b_init := TRUE;
		END_IF

		(*-----------------------Weiterschaltbedingungen----------------------------*)
		IF	haspel_kontroller.st_ctrl.out.b_bereit AND
			rasterfolienmontage.st_ctrl.out.b_bereit AND
			balluff_tag_reader.st_ctrl.out.b_bereit AND
			edit_mfps.st_ctrl.out.b_bereit
			THEN
				haspel_kontroller.st_ctrl.in.b_init := FALSE;
				stueckzahlen.st_ctrl.in.b_init := FALSE;
				balluff_tag_reader.st_ctrl.in.b_init := FALSE;
				rasterfolienmontage.st_ctrl.in.b_init := FALSE;
				edit_mfps.st_ctrl.in.b_init := FALSE;
				fb_state_entry.i16_next_step := 30;
		END_IF

(*=======================================================*)
	30:
		IF fb_state_entry.E THEN
			rasterfolieneinzug.st_ctrl.in.b_init := TRUE;
		END_IF

		(*-----------------------Weiterschaltbedingungen----------------------------*)
		IF rasterfolieneinzug.st_ctrl.out.b_bereit THEN
			rasterfolieneinzug.st_ctrl.in.b_init := FALSE;
			fb_state_entry.i16_next_step := 40;
		END_IF

(*=======================================================*)
	40:
		IF fb_state_entry.E THEN
			axis_bestueckachse.st_ctrl.in.b_init := TRUE;
		END_IF

		(*-----------------------Weiterschaltbedingungen----------------------------*)
		IF axis_bestueckachse.st_ctrl.out.b_bereit  THEN
			axis_bestueckachse.st_ctrl.in.b_init := FALSE;
			fb_state_entry.i16_next_step := 50;
		END_IF

(*=======================================================*)
	50:
		IF fb_state_entry.E THEN
			axis_z_achse.st_ctrl.in.b_init := TRUE;
			axis_y_achse.st_ctrl.in.b_init := TRUE;
		END_IF

		(*-----------------------Weiterschaltbedingungen----------------------------*)
		IF axis_z_achse.st_ctrl.out.b_bereit AND axis_y_achse.st_ctrl.out.b_bereit THEN
			axis_z_achse.st_ctrl.in.b_init := FALSE;
			axis_y_achse.st_ctrl.in.b_init := FALSE;
			fb_state_entry.i16_next_step := 60;
		END_IF

(*=======================================================*)
	60:
		IF fb_state_entry.E THEN
			axis_virt_master.st_ctrl.in.b_init := TRUE;
		END_IF

		(*-----------------------Weiterschaltbedingungen----------------------------*)
		IF axis_virt_master.st_ctrl.out.b_bereit  THEN
			axis_virt_master.st_ctrl.in.b_init := FALSE;
			fb_state_entry.i16_next_step := 70;
		END_IF

(*=======================================================*)
	70:
		IF fb_state_entry.E THEN
			hublift_links.st_ctrl.in.b_init := TRUE;
			hublift_rechts.st_ctrl.in.b_init := TRUE;
			wt_transport_kontroller.st_ctrl.in.b_init := TRUE;
			ST_TouchProbe.st_ctrl_in.b_init := TRUE;
		END_IF

		(*-----------------------Weiterschaltbedingungen----------------------------*)
		IF 	hublift_links.st_ctrl.out.b_bereit AND
			hublift_rechts.st_ctrl.out.b_bereit AND
			wt_transport_kontroller.st_ctrl.out.b_bereit AND
			ST_TouchProbe.st_ctrl_out.b_bereit
			THEN
				hublift_links.st_ctrl.in.b_init := FALSE;
				hublift_rechts.st_ctrl.in.b_init := FALSE;
				wt_transport_kontroller.st_ctrl.in.b_init := FALSE;
				ST_TouchProbe.st_ctrl_in.b_init := FALSE;
				fb_state_entry.i16_next_step := BEREIT;
		END_IF

(*=======================================================*)
	BEREIT:
		IF fb_state_entry.E THEN
			ST_TippTasten.b_initialisierungsphase  := FALSE;

			(* Setze Maschinenstatus *)
			bm_Maschine_in_Gst := TRUE;
		END_IF

		(*Beim Einfädeln muss der Status geändert werden, damit nicht
		ständig neue Maschinendaten erzeugt werden*)
		IF ST_TippTasten.b_einfaedeln_aktiv THEN
			gi16_maschinenstatusinfo := STATUS_MASCHINE_ARBEITET;
		ELSE
			gi16_maschinenstatusinfo := STATUS_BETRIEBSBEREIT;
		END_IF

		(*-----------------------Weiterschaltbedingungen----------------------------*)
		IF NOT wt_transport_kontroller.st_ctrl.out.b_fertig THEN
			bm_Maschine_in_Gst := FALSE;
			fb_state_entry.i16_next_step := 110;
		END_IF

(*=======================================================*)
	110: (* Produktion *)
		IF fb_state_entry.E THEN
			gi16_maschinenstatusinfo := STATUS_MASCHINE_ARBEITET;
		END_IF

		(*-----------------------Weiterschaltbedingungen----------------------------*)
		IF wt_transport_kontroller.st_ctrl.out.b_fertig THEN
			fb_state_entry.i16_next_step := BEREIT;
		END_IF

(*=======================================================*)
	FEHLER:
		IF fb_state_entry.E THEN
			gi16_maschinenstatusinfo := STATUS_FEHLER;
			bm_Maschine_in_Gst := FALSE;
			ST_TippTasten.b_initialisierungsphase  := FALSE;
			fb_ton_quitt.IN := FALSE;
			s_alte_artikelnummer := '';

			(* Schlecht Stueckzahl erhöhen *)
			IF fb_state_entry.i16_last_step = 110 THEN
				stueckzahlen.st_ctrl.in.b_schlechtteil_produziert := TRUE;
			END_IF

			betriebsfreigaben.st_ctrl.in.b_quitt := FALSE;
			safety.st_ctrl.in.b_quitt := FALSE;
			rasterfolienmontage.st_ctrl.in.b_quitt := FALSE;
			rasterfolieneinzug.st_ctrl.in.b_quitt := FALSE;
			axis_virt_master.st_ctrl.in.b_quitt := FALSE;
			axis_bestueckachse.st_ctrl.in.b_quitt := FALSE;
			axis_y_achse.st_ctrl.in.b_quitt := FALSE;
			axis_z_achse.st_ctrl.in.b_quitt := FALSE;
			ST_TouchProbe.st_ctrl_in.b_quitt := FALSE;
			haspel_kontroller.st_ctrl.in.b_quitt := FALSE;
			hublift_links.st_ctrl.in.b_quitt := FALSE;
			hublift_rechts.st_ctrl.in.b_quitt := FALSE;
			wt_transport_kontroller.st_ctrl.in.b_quitt := FALSE;
			stueckzahlen.st_ctrl.in.b_quitt := FALSE;
			balluff_tag_reader.st_ctrl.in.b_quitt := FALSE;
			bbgen.st_ctrl.in.b_quitt := FALSE;
			edit_mfps.st_ctrl.in.b_quitt := FALSE;
			routing_backpanel.st_ctrl.in.b_quitt := FALSE;
			routing_nachbarpc.st_ctrl.in.b_quitt := FALSE;
			Lesen_Schreiben_Tag.st_ctrl.in.b_quitt := FALSE;
			Service.st_ctrl.in.b_quitt := FALSE;

			axis_virt_master.st_ctrl.in.b_preinit := FALSE;
			axis_bestueckachse.st_ctrl.in.b_preinit := FALSE;
			axis_y_achse.st_ctrl.in.b_preinit := FALSE;
			axis_z_achse.st_ctrl.in.b_preinit := FALSE;

			rasterfolienmontage.st_ctrl.in.b_init := FALSE;
			rasterfolieneinzug.st_ctrl.in.b_init := FALSE;
			axis_virt_master.st_ctrl.in.b_init := FALSE;
			axis_bestueckachse.st_ctrl.in.b_init := FALSE;
			axis_y_achse.st_ctrl.in.b_init := FALSE;
			axis_z_achse.st_ctrl.in.b_init := FALSE;
			ST_TouchProbe.st_ctrl_in.b_init := FALSE;
			haspel_kontroller.st_ctrl.in.b_init := FALSE;
			hublift_links.st_ctrl.in.b_init := FALSE;
			hublift_rechts.st_ctrl.in.b_init := FALSE;
			wt_transport_kontroller.st_ctrl.in.b_init := FALSE;
			stueckzahlen.st_ctrl.in.b_init := FALSE;
			balluff_tag_reader.st_ctrl.in.b_init := FALSE;
			edit_mfps.st_ctrl.in.b_init := FALSE;
		END_IF

		(* Fehlerhandling: was soll bei welchem Fehler passieren? *)
		IF 	NOT fb_ton_quitt.IN THEN
			(* Stoppe/Halte Komponenten an *)
			rasterfolienmontage.st_ctrl.in.b_stop := TRUE;
			rasterfolieneinzug.st_ctrl.in.b_stop := TRUE;
			hublift_links.st_ctrl.in.b_stop := TRUE;
			hublift_rechts.st_ctrl.in.b_stop := TRUE;
			wt_transport_kontroller.st_ctrl.in.b_stop := TRUE;
			stueckzahlen.st_ctrl.in.b_stop := TRUE;
			balluff_tag_reader.st_ctrl.in.b_stop := TRUE;
			edit_mfps.st_ctrl.in.b_stop := TRUE;

			(* Diese Fehler führt zum "Stop" in der Maschine *)
			IF safety.st_ctrl.out.b_fehler THEN
				axis_virt_master.st_ctrl.in.b_stop := TRUE;
				axis_bestueckachse.st_ctrl.in.b_stop := TRUE;
				axis_z_achse.st_ctrl.in.b_stop := TRUE;
				axis_y_achse.st_ctrl.in.b_stop := TRUE;
				axis_virt_master.st_ctrl.in.b_halt := FALSE;
				axis_bestueckachse.st_ctrl.in.b_halt := FALSE;
				axis_z_achse.st_ctrl.in.b_halt := FALSE;
				axis_y_achse.st_ctrl.in.b_halt := FALSE;
			ELSE
				axis_virt_master.st_ctrl.in.b_halt := TRUE;
				axis_bestueckachse.st_ctrl.in.b_halt := TRUE;
				axis_z_achse.st_ctrl.in.b_halt := TRUE;
				axis_y_achse.st_ctrl.in.b_halt := TRUE;
				axis_virt_master.st_ctrl.in.b_stop := FALSE;
				axis_bestueckachse.st_ctrl.in.b_stop := FALSE;
				axis_z_achse.st_ctrl.in.b_stop := FALSE;
				axis_y_achse.st_ctrl.in.b_stop := FALSE;
			END_IF
		END_IF


		(*-----------------------Weiterschaltbedingungen----------------------------*)
		IF fb_r_trig_quittieren.Q THEN
			fb_ton_wz.IN:=TRUE;
			b_Merker_quitt:=TRUE;
		END_IF
		IF 	(b_Merker_quitt AND ST_Betriebsfreigaben.e_druckwaechter) OR
			fb_ton_wz.Q THEN
			fb_ton_wz.IN:=FALSE;
			b_Merker_quitt:=FALSE;
			fb_ton_quitt.IN := TRUE;
			(* QUITT *)
			betriebsfreigaben.st_ctrl.in.b_quitt := TRUE;
			safety.st_ctrl.in.b_quitt := TRUE;
			rasterfolienmontage.st_ctrl.in.b_quitt := TRUE;
			rasterfolieneinzug.st_ctrl.in.b_quitt := TRUE;
			axis_virt_master.st_ctrl.in.b_quitt := TRUE;
			axis_bestueckachse.st_ctrl.in.b_quitt := TRUE;
			axis_y_achse.st_ctrl.in.b_quitt := TRUE;
			axis_z_achse.st_ctrl.in.b_quitt := TRUE;
			ST_TouchProbe.st_ctrl_in.b_quitt := TRUE;
			haspel_kontroller.st_ctrl.in.b_quitt := TRUE;
			hublift_links.st_ctrl.in.b_quitt := TRUE;
			hublift_rechts.st_ctrl.in.b_quitt := TRUE;
			wt_transport_kontroller.st_ctrl.in.b_quitt := TRUE;
			stueckzahlen.st_ctrl.in.b_quitt := TRUE;
			balluff_tag_reader.st_ctrl.in.b_quitt := TRUE;
			bbgen.st_ctrl.in.b_quitt := TRUE;
			edit_mfps.st_ctrl.in.b_quitt := TRUE;
			routing_backpanel.st_ctrl.in.b_quitt := TRUE;
			routing_nachbarpc.st_ctrl.in.b_quitt := TRUE;
			Lesen_Schreiben_Tag.st_ctrl.in.b_quitt := TRUE;
			Service.st_ctrl.in.b_quitt := TRUE;
			(* STOP *)
			rasterfolienmontage.st_ctrl.in.b_stop := FALSE;
			rasterfolieneinzug.st_ctrl.in.b_stop := FALSE;
			axis_virt_master.st_ctrl.in.b_stop := FALSE;
			axis_bestueckachse.st_ctrl.in.b_stop := FALSE;
			axis_y_achse.st_ctrl.in.b_stop := FALSE;
			axis_z_achse.st_ctrl.in.b_stop := FALSE;
			haspel_kontroller.st_ctrl.in.b_stop := FALSE;
			hublift_links.st_ctrl.in.b_stop := FALSE;
			hublift_rechts.st_ctrl.in.b_stop := FALSE;
			wt_transport_kontroller.st_ctrl.in.b_stop := FALSE;
			stueckzahlen.st_ctrl.in.b_stop := FALSE;
			balluff_tag_reader.st_ctrl.in.b_stop := FALSE;
			edit_mfps.st_ctrl.in.b_stop := FALSE;
			(* HALT - nur Achsen *)
			axis_virt_master.st_ctrl.in.b_halt := FALSE;
			axis_bestueckachse.st_ctrl.in.b_halt := FALSE;
			axis_y_achse.st_ctrl.in.b_halt := FALSE;
			axis_z_achse.st_ctrl.in.b_halt := FALSE;
		END_IF

		IF fb_ton_quitt.Q THEN
			IF (gi16_betriebsart = AUTO OR gi16_betriebsart = TIPPEN) THEN
				fb_state_entry.i16_next_step := INIT;
			END_IF
		END_IF
END_CASE

fb_state_entry(
	i16_next_step:= ,
	i16_pos:= 2,
	s_debugtext:= ,
	E=> ,
	X=> , 
	i16_step=> ,
	i16_last_step=> );

IF st_config.b_config_fertig THEN
	(* Fehlermeldungen und Betriebsmeldungen ab dem Startindex in die globalen Meldungsarrays schreiben *)
	garr_stoermeldungen[st_config.i16_meld_startindex + 0] := FALSE;
	garr_stoermeldungen[st_config.i16_meld_startindex + 1] := FALSE;
	garr_stoermeldungen[st_config.i16_meld_startindex + 2] := FALSE;
	garr_stoermeldungen[st_config.i16_meld_startindex + 3] := FALSE;
	garr_stoermeldungen[st_config.i16_meld_startindex + 4] := FALSE;
	garr_stoermeldungen[st_config.i16_meld_startindex + 5] := FALSE;
	garr_stoermeldungen[st_config.i16_meld_startindex + 6] := FALSE;
	garr_stoermeldungen[st_config.i16_meld_startindex + 7] := FALSE;
	garr_stoermeldungen[st_config.i16_meld_startindex + 8] := FALSE;
	garr_stoermeldungen[st_config.i16_meld_startindex + 9] := FALSE;
	garr_stoermeldungen[st_config.i16_meld_startindex + 10] := FALSE;
	garr_stoermeldungen[st_config.i16_meld_startindex + 11] := FALSE;
	garr_stoermeldungen[st_config.i16_meld_startindex + 12] := FALSE;
	garr_stoermeldungen[st_config.i16_meld_startindex + 13] := FALSE;
	garr_stoermeldungen[st_config.i16_meld_startindex + 14] := FALSE;
	garr_stoermeldungen[st_config.i16_meld_startindex + 15] := FALSE;
	garr_stoermeldungen[st_config.i16_meld_startindex + 16] := FALSE;
	garr_stoermeldungen[st_config.i16_meld_startindex + 17] := FALSE;
	garr_stoermeldungen[st_config.i16_meld_startindex + 18] := FALSE;
	garr_stoermeldungen[st_config.i16_meld_startindex + 19] := FALSE;
	
	garr_betriebsmeldungen[st_config.i16_meld_startindex + 0] := bm_Maschine_in_Gst;
	garr_betriebsmeldungen[st_config.i16_meld_startindex + 1] := FALSE;
	garr_betriebsmeldungen[st_config.i16_meld_startindex + 2] := FALSE;
	garr_betriebsmeldungen[st_config.i16_meld_startindex + 3] := FALSE;
	garr_betriebsmeldungen[st_config.i16_meld_startindex + 4] := FALSE;
	garr_betriebsmeldungen[st_config.i16_meld_startindex + 5] := FALSE;
	garr_betriebsmeldungen[st_config.i16_meld_startindex + 6] := FALSE;
	garr_betriebsmeldungen[st_config.i16_meld_startindex + 7] := FALSE;
	garr_betriebsmeldungen[st_config.i16_meld_startindex + 8] := FALSE;
	garr_betriebsmeldungen[st_config.i16_meld_startindex + 9] := FALSE;
	garr_betriebsmeldungen[st_config.i16_meld_startindex + 10] := FALSE;
	garr_betriebsmeldungen[st_config.i16_meld_startindex + 11] := FALSE;
	garr_betriebsmeldungen[st_config.i16_meld_startindex + 12] := FALSE;
	garr_betriebsmeldungen[st_config.i16_meld_startindex + 13] := FALSE;
	garr_betriebsmeldungen[st_config.i16_meld_startindex + 14] := FALSE;
	garr_betriebsmeldungen[st_config.i16_meld_startindex + 15] := FALSE;
	garr_betriebsmeldungen[st_config.i16_meld_startindex + 16] := FALSE;
	garr_betriebsmeldungen[st_config.i16_meld_startindex + 17] := FALSE;
	garr_betriebsmeldungen[st_config.i16_meld_startindex + 18] := FALSE;
	garr_betriebsmeldungen[st_config.i16_meld_startindex + 19] := FALSE;
END_IF
END_PROGRAM

(* POU Maschine1700/Einpresskraftueberwachung/ST_Einpress_Kontroller_alt, ST *)
PROGRAM ST_Einpress_Kontroller_alt
VAR_INPUT
	st_config									: struct_config;
	st_ctrl_in									: struct_ctrl_in;
	lr_achsposition							: LREAL;
END_VAR
VAR_IN_OUT
	st_visu									: struct_visu;
	st_einpressen							: struct_einpresskraftueberwachung;
END_VAR
VAR_OUTPUT
	st_ctrl_out								: struct_ctrl_out;
END_VAR
VAR
	fb_ton_wz								: TON;
	fb_ton_uez								: TON;
	fb_ton_quitt								: TON;
	fb_r_trig_start								: R_TRIG;
	fb_state_entry								: ST_StateEntry;
	lr_kraft_n									: LREAL := 0.0;
	lr_weg_grad								: LREAL := 0.0;
	i16_pin_nr								: INT := 0;
	i16_kraftfaktor								: INT := 0;
	ui_akt_pos_bestueckachse					: UINT := 0;
	i16_ku_nr								: INT := 0;
	i16_mp_nr								: INT := 0;
	b_kraft_weg_in_mp_ok						: BOOL := FALSE;
	sm_fehler_einpressmodus					: BOOL := FALSE;
	sm_aktkraft_groesser_maxkraft_aufnahme	: BOOL := FALSE;
	sm_aktkraft_groesser_maxkraft_einpressen	: BOOL := FALSE;
	sm_aktkraft_kleiner_minkraft_einpressen		: BOOL := FALSE;
	sm_kraft_weg_ausserhalb_huellkurve		: BOOL := FALSE;
	sm_fehler_analogwert_kraftmessdose		: BOOL := FALSE;
	sm_max_mb_ueberschritten					: BOOL := FALSE;
	sm_max_einstell_mb_ueberschritten			: BOOL := FALSE;

	a_start_messung							AT %Q* : BOOL := FALSE;
	a_messbereich_1_oder_2					AT %Q* : BOOL := FALSE;	(* MB1 = low, MB2 = high *)

	st_ausgabe								: struct_einpressausgabe;
	i16_merker								: INT := 0;
	lr_help_maxkraft_einpressen				:LREAL;
END_VAR
VAR CONSTANT
	i_KRAFTFAKTOR_MB1		: INT := 200;	(* Der Kraftfaktor richtet sich nach der Messbereichskalibrierung in der Zusatzsoftware (ICAM) für den Ladungsverstärker *)
	i_KRAFTFAKTOR_MB2		: INT := 2000;
	i_MAX_MESSPUNKTE			: INT := 360;
	i_MAX_KURVEN				: INT := 99;
END_VAR
(* Zeiten *)
fb_ton_wz(IN:= , PT:= , Q=>  , ET=> );
fb_ton_uez(IN:= , PT:= , Q=>  , ET=> );

fb_ton_quitt(IN:= , PT:= t#100ms, Q=> , ET=> );

(* Flanken *)
fb_r_trig_start(CLK:= st_ctrl_in.b_start, Q=> );

(* Analogwert Kraftmessdose *)
kraftmessdose.fb(
	t_verzoegerung:= t#500ms,
	st_config:= kraftmessdose.fb.st_config);

(* Berechnung der aktuellen Kraft in Newton aus dem Analogwert in  Volt. *)
(* Die Normierung der Analogspannung als Kraft erfolgt mit dem Kalibrierschein der Kraftmessdose und der Software "ICAM5073" *)
(* Eingestellter Messbereich1: 0 - 200N, Messbereich2: 0 - 2000N *)
IF a_messbereich_1_oder_2 THEN
	i16_kraftfaktor := i_KRAFTFAKTOR_MB2;
ELSE
	i16_kraftfaktor := i_KRAFTFAKTOR_MB1;
END_IF

(* nur bei voller Drehzahl mit eingestellter Kraft prüfen*)
IF	ST_TippTasten.i16_akt_stufe = 9 THEN
	lr_help_maxkraft_einpressen:=st_einpressen.st_einstellungen.lr_maxkraft_einpressen;
ELSE
	lr_help_maxkraft_einpressen:=800;
END_IF

(* Behandlung Ausnahmefall Division durch 0  *)
IF kraftmessdose.fb.i16_anzeigewert_max <> 0 THEN
	lr_kraft_n := i16_kraftfaktor * kraftmessdose.fb.st_sensor.e_i16_value / kraftmessdose.fb.i16_anzeigewert_max;
END_IF

lr_weg_grad := lr_achsposition;
ui_akt_pos_bestueckachse := LREAL_TO_UINT(lr_achsposition);

(* ===============Toplevel================ *)
IF fb_state_entry.i16_next_step > INIT AND fb_state_entry.i16_next_step < FEHLER THEN
	IF fb_state_entry.i16_next_step < STOP THEN
		IF st_ctrl_in.b_stop THEN
			fb_state_entry.i16_next_step := STOP;
		END_IF
	END_IF

	(* Fehlersignal der Kraftmessdose *)
	IF st_config.b_station_aktiv THEN
		IF kraftmessdose.fb.b_error THEN
			sm_fehler_analogwert_kraftmessdose := TRUE;
			fb_state_entry.i16_next_step := FEHLER;
		END_IF
		IF 	(NOT a_messbereich_1_oder_2 AND lr_kraft_n > i_KRAFTFAKTOR_MB1) OR
			(a_messbereich_1_oder_2 AND lr_kraft_n > i_KRAFTFAKTOR_MB2) OR
			(gst_datensatz.st_band.st_einpressen.st_einstellungen.lr_maxkraft_einpressen > i_KRAFTFAKTOR_MB2)
			THEN
				sm_max_mb_ueberschritten := TRUE;
				fb_state_entry.i16_next_step := FEHLER;
		END_IF
		IF gst_datensatz.st_band.st_einpressen.st_einstellungen.lr_maxkraft_einpressen > i_KRAFTFAKTOR_MB2 THEN
			sm_max_einstell_mb_ueberschritten := TRUE;
			fb_state_entry.i16_next_step := FEHLER;
		END_IF
	END_IF
END_IF

(* ======================================Schrittkette======================================== *)
fb_state_entry(
	i16_next_step:= ,
	i16_pos:= 1,
	s_debugtext:= ,
	E=> ,
	X=> ,
	i16_step=> ,
	i16_last_step=> );

CASE fb_state_entry.i16_step OF
(*=======================================================*)
	INIT_OBJ:
		IF st_config.b_config_fertig THEN
			a_messbereich_1_oder_2 := FALSE;
			fb_state_entry.i16_next_step := INIT;
		END_IF

(*=======================================================*)
	INIT:
		IF fb_state_entry.E THEN
			fb_ton_wz.IN := FALSE;
			fb_ton_uez.IN := FALSE;
			fb_ton_quitt.IN := FALSE;
			st_ctrl_out.b_fehler := FALSE;
			st_ctrl_out.b_bereit := FALSE;
			st_ctrl_out.b_fertig := FALSE;
			a_start_messung := FALSE;
			i16_pin_nr := 0;
			sm_fehler_einpressmodus := FALSE;
			sm_aktkraft_groesser_maxkraft_aufnahme := FALSE;
			sm_aktkraft_groesser_maxkraft_einpressen := FALSE;
			sm_aktkraft_kleiner_minkraft_einpressen := FALSE;
			sm_kraft_weg_ausserhalb_huellkurve := FALSE;
			sm_fehler_analogwert_kraftmessdose := FALSE;
			sm_max_mb_ueberschritten := FALSE;
			sm_max_einstell_mb_ueberschritten := FALSE;
		END_IF

		(*-----------------------Weiterschaltbedingungen----------------------------*)
		IF st_ctrl_in.b_init THEN
			fb_state_entry.i16_next_step := BEREIT;
		END_IF

(*=======================================================*)
	BEREIT:
		IF fb_state_entry.E THEN
			st_ctrl_out.b_bereit := TRUE;
			st_ctrl_out.b_fertig := TRUE;
			i16_pin_nr := 0;
		END_IF

		(*-----------------------Weiterschaltbedingungen----------------------------*)
		IF st_ctrl_in.b_start THEN
			fb_state_entry.i16_next_step := 110;
		END_IF

(*=======================================================*)
	110:	(* Kraftmessung starten *)
		IF fb_state_entry.E THEN
			st_ctrl_out.b_fertig := FALSE;
			a_start_messung := TRUE;
			st_ausgabe.st_ergebnisse.lr_maxkraft_einpressen := 0;
			st_ausgabe.st_ergebnisse.lr_maxkraft_einpres_proHub:=0;
			st_ausgabe.st_ergebnisse.lr_ueberlaufkraft := 0;

